(* CODESYS project PCL_CoralP

Project tree, tasks and I/O mapping:
  Device : CODESYS Control for Linux SL, CODESYS, order no. 2302000005, version 4.11.0.0
    Ethernet : Ethernet, CODESYS, version 4.2.0.0
        settings: IPAddress = [172,16,0,11]; SubnetMask = [205,255,255,0]; GatewayAddress = [0,0,0,0]; MACAddress = [16#00,16#E0,16#4F,16#68,16#EC,16#4A]; NetworkInterfaceName = 'eno1'; NetworkInterfaceName = "eno1"; SaveCommunicationSettings = FALSE; IPAddress = [192,168,0,2]; SubnetMask = [255,255,255,0]; GatewayAddress = [0,0,0,0]
      Modbus_TCP_Master : Modbus TCP Master, 3S - Smart Software Solutions GmbH, version 4.3.0.0 (disabled)
          settings: AutoReconnect = TRUE
        Modbus_TCP_Slave_AC1 : Modbus TCP Slave, 3S - Smart Software Solutions GmbH, version 4.1.0.0
            settings: Unit-ID = 255; IPAddress = [192, 168, 0, 51]; Channel 0.Function Code = 3; Channel 0.Read Offset = 16#0000; Channel 0.Read Length = 124; Channel 0.Write Offset = 0; Channel 0.Write Length = 0; Channel 0.Cycle Time = 100; Channel 1.Function Code = 3; Channel 1.Read Offset = 16#007C; Channel 1.Read Length = 124; Channel 1.Write Offset = 0; Channel 1.Write Length = 0; Channel 1.Cycle Time = 100; Channel 2.Function Code = 3; Channel 2.Read Offset = 16#00F8; Channel 2.Read Length = 124; Channel 2.Write Offset = 0; Channel 2.Write Length = 0; Channel 2.Cycle Time = 100; Channel 3.Function Code = 16; Channel 3.Read Offset = 0; Channel 3.Read Length = 0; Channel 3.Write Offset = 16#0114; Channel 3.Write Length = 4; Channel 3.Cycle Time = 100
            output Application.Chiller_1.modbus_var_1002[276] : WORD  // Channel 3.Channel 3
            output Application.Chiller_1.modbus_var_1002[277] : WORD  // Channel 3.Channel 3
            output Application.Chiller_1.modbus_var_1002[278] : WORD  // Channel 3.Channel 3
            output Application.Chiller_1.modbus_var_1002[279] : WORD  // Channel 3.Channel 3
            unmapped channels: Channel 0, Channel 1, Channel 2, Channel 3
  Modbus_Master_COM_Port_1 : Modbus Master, COM Port, 3S - Smart Software Solutions GmbH, version 4.3.0.0
      settings: Auto-restart communication = TRUE
    Modbus_Server_COM_Port_AC1 : Modbus Server, COM Port, CODESYS, version 4.4.0.0
        settings: SlaveAddress = 18; ResponseTimeout = 1000; UseExtendedFunctionCodes = TRUE; Channel 0.Function Code = 3; Channel 0.Read Offset = 16#0000; Channel 0.Read Length = 91; Channel 0.Write Offset = 0; Channel 0.Write Length = 0; Channel 0.Cycle Time = 100
        input  Application.Chiller_1.modbus_var_1000 : ARRAY[0..90] OF WORD  // Channel 0
    Modbus_Server_COM_Port_AC2 : Modbus Server, COM Port, CODESYS, version 4.4.0.0
        settings: SlaveAddress = 18; ResponseTimeout = 1000; UseExtendedFunctionCodes = TRUE; Channel 0.Function Code = 3; Channel 0.Read Offset = 16#0000; Channel 0.Read Length = 91; Channel 0.Write Offset = 0; Channel 0.Write Length = 0; Channel 0.Cycle Time = 100
        input  Application.Chiller_2.modbus_var_1000 : ARRAY[0..90] OF WORD  // Channel 0
    Modbus_Slave_COM_Port_AC1 : Modbus Slave, COM Port, 3S - Smart Software Solutions GmbH, version 4.1.0.0
        settings: SlaveAddress = 18; ResponseTimeout = 1000; UseExtendedFunctionCodes = TRUE; Channel 0.Function Code = 3; Channel 0.Read Offset = 16#0000; Channel 0.Read Length = 100; Channel 0.Write Offset = 0; Channel 0.Write Length = 0; Channel 0.Cycle Time = 100
        input  Application.Chiller_1.modbus_var_1000 : ARRAY[0..99] OF WORD  // Channel 0
    Modbus_Slave_COM_Port_AC2 : Modbus Slave, COM Port, 3S - Smart Software Solutions GmbH, version 4.1.0.0
        settings: SlaveAddress = 18; ResponseTimeout = 1000; UseExtendedFunctionCodes = TRUE; Channel 0.Function Code = 3; Channel 0.Read Offset = 16#0200; Channel 0.Read Length = 91; Channel 0.Write Offset = 0; Channel 0.Write Length = 0; Channel 0.Cycle Time = 100
        input  Application.Chiller_2.modbus_var_1000 : ARRAY[0..90] OF WORD  // Channel 0
    Modbus_Slave_COM_Port_AC3 : Modbus Slave, COM Port, 3S - Smart Software Solutions GmbH, version 4.1.0.0
        settings: SlaveAddress = 18; ResponseTimeout = 1000; UseExtendedFunctionCodes = TRUE; Channel 0.Function Code = 3; Channel 0.Read Offset = 16#0400; Channel 0.Read Length = 91; Channel 0.Write Offset = 0; Channel 0.Write Length = 0; Channel 0.Cycle Time = 100
        input  Application.Chiller_3.modbus_var_1000 : ARRAY[0..90] OF WORD  // Channel 0
    Modbus_Slave_COM_Port_AC4 : Modbus Slave, COM Port, 3S - Smart Software Solutions GmbH, version 4.1.0.0
        settings: SlaveAddress = 18; ResponseTimeout = 1000; UseExtendedFunctionCodes = TRUE; Channel 0.Function Code = 3; Channel 0.Read Offset = 16#0600; Channel 0.Read Length = 91; Channel 0.Write Offset = 0; Channel 0.Write Length = 0; Channel 0.Cycle Time = 100
        input  Application.Chiller_4.modbus_var_1000 : ARRAY[0..90] OF WORD  // Channel 0
    Modbus_Slave_COM_Seq : Modbus Slave, COM Port, 3S - Smart Software Solutions GmbH, version 4.1.0.0
        settings: SlaveAddress = 18; ResponseTimeout = 1000; UseExtendedFunctionCodes = TRUE; Channel 0.Function Code = 3; Channel 0.Read Offset = 16#0A00; Channel 0.Read Length = 125; Channel 0.Write Offset = 0; Channel 0.Write Length = 0; Channel 0.Cycle Time = 100; Channel 1.Function Code = 3; Channel 1.Read Offset = 16#0A7D; Channel 1.Read Length = 34; Channel 1.Write Offset = 0; Channel 1.Write Length = 0; Channel 1.Cycle Time = 100; Channel 2.Function Code = 16; Channel 2.Read Offset = 0; Channel 2.Read Length = 0; Channel 2.Write Offset = 16#0A8B; Channel 2.Write Length = 4; Channel 2.Cycle Time = 100; Channel 3.Function Code = 16; Channel 3.Read Offset = 0; Channel 3.Read Length = 0; Channel 3.Write Offset = 16#0A95; Channel 3.Write Length = 4; Channel 3.Cycle Time = 100
        input  Application.Sequence.modbus_var_1000 : ARRAY[0..124] OF WORD  // Channel 0
        input  Application.Sequence.modbus_var_1001 : ARRAY[0..33] OF WORD  // Channel 1
        output Application.Sequence.modbus_var_PI : ARRAY[0..3] OF WORD  // Channel 2
        output Application.Sequence.modbus_var_wasted : ARRAY[0..3] OF WORD  // Channel 3
  libraries: CmpBitmapPool, 3.5.17.0 (System); AC_DataLog, 3.5.16.0 (3S - Smart Software Solutions GmbH)
  5ce3da45-db07-42e7-a21c-a00fff4ed8f6|C:\Users\Codesys\Desktop\Images\Div bilder\Arrow gray left.png
  5ce3da45-db07-42e7-a21c-a00fff4ed8f6|C:\Users\Codesys\Desktop\Images\Div bilder\Arrow green down.png
  5ce3da45-db07-42e7-a21c-a00fff4ed8f6|C:\Users\Codesys\Desktop\Images\Div bilder\Arrow green up.png
  5ce3da45-db07-42e7-a21c-a00fff4ed8f6|C:\Users\Codesys\Desktop\Images\Div bilder\Arrow lightblue left.png
  5ce3da45-db07-42e7-a21c-a00fff4ed8f6|C:\Users\Codesys\Desktop\Images\Div bilder\Arrow red down.png
  5ce3da45-db07-42e7-a21c-a00fff4ed8f6|C:\Users\Codesys\Desktop\Images\Div bilder\Arrow red left.png
  5ce3da45-db07-42e7-a21c-a00fff4ed8f6|C:\Users\Codesys\Desktop\Images\Invisible.png
  5ce3da45-db07-42e7-a21c-a00fff4ed8f6|C:\Users\Codesys\Desktop\Images\LEDS\ALARM.png
  5ce3da45-db07-42e7-a21c-a00fff4ed8f6|C:\Users\Codesys\Desktop\Images\LEDS\Led_SQ_Green1_On_Medium.png
  5ce3da45-db07-42e7-a21c-a00fff4ed8f6|C:\Users\Codesys\Desktop\Images\LEDS\Led_SQ_Grey_Off_Medium.png
  5ce3da45-db07-42e7-a21c-a00fff4ed8f6|C:\Users\Codesys\Desktop\Images\LEDS\TRIP.png
  5ce3da45-db07-42e7-a21c-a00fff4ed8f6|C:\Users\Codesys\Desktop\Images\Logo-Aida.png
  5ce3da45-db07-42e7-a21c-a00fff4ed8f6|C:\Users\Codesys\Desktop\Images\Logo-Costa.png
  5ce3da45-db07-42e7-a21c-a00fff4ed8f6|C:\Users\Codesys\Desktop\Images\Logo-HAL.png
  5ce3da45-db07-42e7-a21c-a00fff4ed8f6|C:\Users\Codesys\Desktop\Images\Logo-ncl.png
  5ce3da45-db07-42e7-a21c-a00fff4ed8f6|C:\Users\Codesys\Desktop\Images\Logo-Princess.png
  5ce3da45-db07-42e7-a21c-a00fff4ed8f6|C:\Users\Codesys\Desktop\Images\Logo-TUI.png
  5ce3da45-db07-42e7-a21c-a00fff4ed8f6|C:\Users\Codesys\Desktop\Images\Menu\AlarmMenu.png
  5ce3da45-db07-42e7-a21c-a00fff4ed8f6|C:\Users\Codesys\Desktop\Images\Pipes\PipeGreen_1_Horizontal.png
  5ce3da45-db07-42e7-a21c-a00fff4ed8f6|C:\Users\Codesys\Desktop\Images\Pipes\PipeGreen_1_LD.png
  5ce3da45-db07-42e7-a21c-a00fff4ed8f6|C:\Users\Codesys\Desktop\Images\Pipes\PipeGreen_2_LU.png
  5ce3da45-db07-42e7-a21c-a00fff4ed8f6|C:\Users\Codesys\Desktop\Images\Pipes\PipeGreen_3way_2.png
  5ce3da45-db07-42e7-a21c-a00fff4ed8f6|C:\Users\Codesys\Desktop\Images\Pipes\PipeGreen_3way.png
  5ce3da45-db07-42e7-a21c-a00fff4ed8f6|C:\Users\Codesys\Desktop\Images\Pipes\PipeGrey_1S_Horizontal.png
  5ce3da45-db07-42e7-a21c-a00fff4ed8f6|C:\Users\Codesys\Desktop\Images\Pipes\PipeGrey_2_LD.png
  5ce3da45-db07-42e7-a21c-a00fff4ed8f6|C:\Users\Codesys\Desktop\Images\Pipes\PipeGrey_3_LU.png
  5ce3da45-db07-42e7-a21c-a00fff4ed8f6|C:\Users\Codesys\Desktop\Images\Pipes\PipeLightBlue_1_Horizontal.png
  5ce3da45-db07-42e7-a21c-a00fff4ed8f6|C:\Users\Codesys\Desktop\Images\Pipes\PipeLightBlue_1_LD.png
  5ce3da45-db07-42e7-a21c-a00fff4ed8f6|C:\Users\Codesys\Desktop\Images\Pipes\PipeLightBlue_1_Vertical.png
  5ce3da45-db07-42e7-a21c-a00fff4ed8f6|C:\Users\Codesys\Desktop\Images\Pipes\PipeLightBlue_2_LU.png
  5ce3da45-db07-42e7-a21c-a00fff4ed8f6|C:\Users\Codesys\Desktop\Images\Pipes\PipeLightBlue_3_RD.png
  5ce3da45-db07-42e7-a21c-a00fff4ed8f6|C:\Users\Codesys\Desktop\Images\Pipes\PipeLightBlue_3_RU.png
  5ce3da45-db07-42e7-a21c-a00fff4ed8f6|C:\Users\Codesys\Desktop\Images\Pipes\PipeRed_1_LD.png
  5ce3da45-db07-42e7-a21c-a00fff4ed8f6|C:\Users\Codesys\Desktop\Images\Pipes\PipeRed_1_RD.png
  5ce3da45-db07-42e7-a21c-a00fff4ed8f6|C:\Users\Codesys\Desktop\Images\Pipes\PipeRed_2_Horizontal.png
  5ce3da45-db07-42e7-a21c-a00fff4ed8f6|C:\Users\Codesys\Desktop\Images\Pipes\PipeRed_2_LU.png
  5ce3da45-db07-42e7-a21c-a00fff4ed8f6|C:\Users\Codesys\Desktop\Images\Pipes\PipeRed_2_RU.png
  5ce3da45-db07-42e7-a21c-a00fff4ed8f6|C:\Users\Codesys\Desktop\Images\Pumps\Pump_Large_3.png
  5ce3da45-db07-42e7-a21c-a00fff4ed8f6|C:\Users\Codesys\Desktop\Images\Scales\BarScale3.png
  5ce3da45-db07-42e7-a21c-a00fff4ed8f6|C:\Users\Codesys\Desktop\Images\Scales\BarScale4.png
  5ce3da45-db07-42e7-a21c-a00fff4ed8f6|C:\Users\Codesys\Desktop\Images\Transparants\CapBarTranparant.png
  5ce3da45-db07-42e7-a21c-a00fff4ed8f6|C:\Users\Codesys\Desktop\Images\Valves\Valve_2.png
  5ce3da45-db07-42e7-a21c-a00fff4ed8f6|C:\Users\Codesys\Desktop\Images\Valves\Valve_3.png
  5ce3da45-db07-42e7-a21c-a00fff4ed8f6|C:\Users\Codesys\Desktop\Images\Valves\Valve_4.png
  5ce3da45-db07-42e7-a21c-a00fff4ed8f6|C:\Users\Codesys\Desktop\MenuAlarm.png
  5ce3da45-db07-42e7-a21c-a00fff4ed8f6|C:\Users\Codesys\Desktop\MenuEvents.png
  5ce3da45-db07-42e7-a21c-a00fff4ed8f6|C:\Users\Codesys\Desktop\MenuHome.png
  5ce3da45-db07-42e7-a21c-a00fff4ed8f6|C:\Users\Codesys\Desktop\MenuLogout.png
  5ce3da45-db07-42e7-a21c-a00fff4ed8f6|C:\Users\Codesys\Desktop\MenuSchematics.png
  5ce3da45-db07-42e7-a21c-a00fff4ed8f6|C:\Users\Codesys\Desktop\MenuSettings.png
  5ce3da45-db07-42e7-a21c-a00fff4ed8f6|C:\Users\Codesys\Desktop\white.PNG
  5ce3da45-db07-42e7-a21c-a00fff4ed8f6|C:\Users\Codesys\Documents\logo\1200px-Johnson_Controls.svg.png
  5ce3da45-db07-42e7-a21c-a00fff4ed8f6|C:\Users\Codesys\Documents\logo\JCI_Full Color_Transparent Background.png
  5ce3da45-db07-42e7-a21c-a00fff4ed8f6|C:\Users\Codesys\Pictures\ConquestVSChiller1.jpg
  5ce3da45-db07-42e7-a21c-a00fff4ed8f6|C:\Users\Codesys\Pictures\Grafic_oldradar\2016_update\Images\Chiller\Compressor.png
  5ce3da45-db07-42e7-a21c-a00fff4ed8f6|C:\Users\Codesys\Pictures\Grafic_oldradar\2016_update\Images\Chiller\Condenser.png
  5ce3da45-db07-42e7-a21c-a00fff4ed8f6|C:\Users\Codesys\Pictures\Grafic_oldradar\2016_update\Images\Chiller\Evaporator.png
  5ce3da45-db07-42e7-a21c-a00fff4ed8f6|C:\Users\Technician\Desktop\Images\Pipes\PipeBlack_1_Vertical.png
  5ce3da45-db07-42e7-a21c-a00fff4ed8f6|C:\Users\Technician\Desktop\Images\Ships\CoralP.jpg
  5ce3da45-db07-42e7-a21c-a00fff4ed8f6|C:\Users\Technician\Desktop\Images\Ships\Diamond.png
  5ce3da45-db07-42e7-a21c-a00fff4ed8f6|C:\Users\Technician\Pictures\C_Sunrise.jpg
  5ce3da45-db07-42e7-a21c-a00fff4ed8f6|C:\Users\Technician\Pictures\Sapphire-princess.jpg
  5ce3da45-db07-42e7-a21c-a00fff4ed8f6|E:\Images\Images\Chiller\ACChiller3D.png
  text list GlobalTextList
  visualisation AC_Plant_Overview
  Alarm Configuration
  visualisation Alarm_list
  program BlinkingAlarm [CFC]
  program Calculus [ST]
  visualisation Chiller1Menu
  visualisation Chiller2Menu
  visualisation Chiller3Menu
  visualisation Chiller4Menu
  program Chiller_1 [ST]
  visualisation Chiller_1_Alarm
  visualisation Chiller_1_Alarm
  visualisation Chiller_1_Flow_Diagram
  visualisation Chiller_1_Oil
  text list Chiller_1_trendvalues
  visualisation Chiller_1_Trip
  visualisation Chiller_1_Trip
  visualisation Chiller_1_Values
  visualisation Chiller_1_Values
  visualisation Chiller_1_VFD
  program Chiller_2 [ST]
  text list Chiller_2_4_trendvalues
  visualisation Chiller_2_Alarm
  visualisation Chiller_2_Alarm
  visualisation Chiller_2_Flow_Diagram
  visualisation Chiller_2_Flow_Diagram
  visualisation Chiller_2_Oil
  visualisation Chiller_2_Trip
  visualisation Chiller_2_Trip
  visualisation Chiller_2_Values
  visualisation Chiller_2_Values
  visualisation Chiller_3_Alarm
  program Chiller_3 [ST]
  visualisation Chiller_3_Flow_Diagram
  visualisation Chiller_3_Flow_Diagram
  visualisation Chiller_3_Oil
  text list Chiller_3_trendvalues
  visualisation Chiller_3_Trip
  program Chiller_4 [ST]
  visualisation Chiller_4_Alarm
  visualisation Chiller_4_Alarm
  visualisation Chiller_4_Oil
  text list Chiller_4_trendvalues
  global variables GVL
  text PersistenceConfig
  text list Sequence_trendvalues
  function block AC_DataLogManager [ST]
*)

// GVL
{attribute 'qualified_only'}
VAR_GLOBAL
	COPcalc_data	: ARRAY[0..2, 0..320] OF STRING(100);
	calc_data		: ARRAY[0..8, 0..80] OF STRING(100) ;
	{attribute 'ac_persist' := 'PersistenceChannel'}
	saCOPDataArray			: ARRAY[0..2, 0..320] OF STRING(100);
	{attribute 'ac_persist' := 'PersistenceChannel'}
	saDataArray			: ARRAY[0..8, 0..80] OF STRING(100);
		{attribute 'ac_persist' := 'PersistenceChannel'}
	saDataArray1			: ARRAY[0..8, 0..80] OF STRING(100);
		{attribute 'ac_persist' := 'PersistenceChannel'}
	saDataArray2		: ARRAY[0..8, 0..80] OF STRING(100);
	initRead : BOOL;
	xRead : BOOL;
	xRead1 : BOOL;
	xRead2 : BOOL;
	xReadCOP : BOOL := FALSE;
	startUp : BOOL;
	presstimer  : TON;
	presstimer2 : TON;
	presstimer3 : TON;
	presstimer4 : TON;
	delaytimer  : TON;
	starttimer1 : BOOL := FALSE  ;
	starttimer2 : BOOL := FALSE  ;
	starttimer3 : BOOL := FALSE  ;
	starttimer4 : BOOL := FALSE  ;
	startdelaytimer : BOOL := FALSE ;
	Startonce : BOOL := FALSE ;
	Startsecond : BOOL := FALSE ;
	{attribute 'ac_persist' := 'PersistenceChannel'}
	PIexpireDate : DATE_AND_TIME := DT#2025-12-30-00:00:00;
	CurrentDate : DATE_AND_TIME ;
	
	
END_VAR

// BlinkingAlarm
PROGRAM BlinkingAlarm
VAR
	TimeOn: TIME:= T#1S;
	TimeOff: TIME:= T#1S;
	Alarm: BOOL;
	TurnOn: BOOL;
		
	Blink_0: BLINK;
	
END_VAR
VAR // added by the converter: edge detectors and wires of the graphical bodies
    _w1, _w2 : BOOL;
END_VAR

TurnOn := _w1;
_w1 := not.Sequence.Alarm_sequence OR not.Chiller_1.Unit_alarm OR not.Chiller_1.Unit_trip OR not.Chiller_2.Unit_alarm OR not.Chiller_2.Unit_trip OR not.Chiller_3.Unit_alarm OR not.Chiller_3.Unit_trip OR not.Chiller_4.Unit_alarm OR not.Chiller_4.Unit_trip;
_w2 := TurnOn AND Blink_0.OUT;
Blink_0(ENABLE := TurnOn, TIMELOW := TimeOff, TIMEHIGH := TimeOn); // BLINK
Alarm := _w2;

END_PROGRAM

// Chiller_2
PROGRAM Chiller_2
VAR

timer2 : standard.ton ;
{attribute 'ac_datalog_set_default_group' := 'DatalogChannel_2'}
instStruct : LogStruct;

modbus_var : ARRAY[0..100] OF INT;
modbus_var_1000 : ARRAY[0..123] OF WORD;
modbus_var_1001 : ARRAY[124..247] OF WORD;
modbus_var_1002 : ARRAY[248..371] OF WORD;
{attribute 'ac_datalog_hysteresis' := '0.2'}
{attribute 'ac_datalog' := 'DatalogChannel_2'}
Temp_chilled_medium_out : REAL;
{attribute 'ac_datalog_hysteresis' := '0.2'}
{attribute 'ac_datalog' := 'DatalogChannel_2'}
Temp_chilled_medium_in : REAL;
{attribute 'ac_datalog_hysteresis' := '0.2'}
{attribute 'ac_datalog' := 'DatalogChannel_2'}
Temp_water_inlet_cond : REAL;
{attribute 'ac_datalog_hysteresis' := '0.2'}
{attribute 'ac_datalog' := 'DatalogChannel_2'}
Press_suction_compr : REAL;
{attribute 'ac_datalog_hysteresis' := '0.5'}
{attribute 'ac_datalog' := 'DatalogChannel_2'}
Press_discharge_compr : REAL;
{attribute 'ac_datalog_hysteresis' := '0.5'}
{attribute 'ac_datalog' := 'DatalogChannel_2'}
Press_oil_receiver : REAL;
{attribute 'ac_datalog_hysteresis' := '0.5'}
{attribute 'ac_datalog' := 'DatalogChannel_2'}
Press_oil_compr : REAL;
{attribute 'ac_datalog_hysteresis' := '0.4'}
{attribute 'ac_datalog' := 'DatalogChannel_2'}
Temp_discharge : REAL;
{attribute 'ac_datalog_hysteresis' := '0.5'}
{attribute 'ac_datalog' := 'DatalogChannel_2'}
Oil_temp_receiver : REAL;
{attribute 'ac_datalog_hysteresis' := '0.5'}
{attribute 'ac_datalog' := 'DatalogChannel_2'}
Max_motor_temp : REAL;
{attribute 'ac_datalog_hysteresis' := '0.2'}
{attribute 'ac_datalog' := 'DatalogChannel_2'}
Temp_motor_bearing_DE : REAL;
{attribute 'ac_datalog_hysteresis' := '0.2'}
{attribute 'ac_datalog' := 'DatalogChannel_2'}
Temp_motor_bearing_NDE : REAL;
{attribute 'ac_datalog_hysteresis' := '4'}
{attribute 'ac_datalog' := 'DatalogChannel_2'}
Motor_current : REAL;
{attribute 'ac_datalog_hysteresis' := '50'}
{attribute 'ac_datalog' := 'DatalogChannel_2'}
Running_hours_comp_unscaled : WORD;
{attribute 'ac_datalog_hysteresis' := '50'}
{attribute 'ac_datalog' := 'DatalogChannel_2'}
Running_hours_oil_pump_unscaled : WORD;
{attribute 'ac_datalog' := 'DatalogChannel_2'}
Anti_recycle_time : REAL;
{attribute 'ac_datalog_hysteresis' := '2'}
{attribute 'ac_datalog' := 'DatalogChannel_2'}
Feedback_compressor : REAL;
{attribute 'ac_datalog_hysteresis' := '0.2'}
{attribute 'ac_datalog' := 'DatalogChannel_2'}
Oil_diff_pressure : REAL;
{attribute 'ac_datalog_hysteresis' := '0.3'}
{attribute 'ac_datalog' := 'DatalogChannel_2'}
Suction_saturated_temp : REAL;
{attribute 'ac_datalog_hysteresis' := '0.2'}
{attribute 'ac_datalog' := 'DatalogChannel_2'}
Discharge_saturated_temp : REAL;
{attribute 'ac_datalog_hysteresis' := '0.2'}
{attribute 'ac_datalog' := 'DatalogChannel_2'}
Temp_water_outlet_cond : REAL;
{attribute 'ac_datalog_hysteresis' := '0.2'}
{attribute 'ac_datalog' := 'DatalogChannel_2'}
Temp_motor_wind_R : REAL;
{attribute 'ac_datalog_hysteresis' := '0.2'}
{attribute 'ac_datalog' := 'DatalogChannel_2'}
Temp_motor_wind_S : REAL;
{attribute 'ac_datalog_hysteresis' := '0.2'}
{attribute 'ac_datalog' := 'DatalogChannel_2'}
Temp_motor_wind_T : REAL;
{attribute 'ac_datalog_hysteresis' := '0.2'}
{attribute 'ac_datalog' := 'DatalogChannel_2'}
Temp_motor_air : REAL;
{attribute 'ac_datalog_hysteresis' := '0.04'}
{attribute 'ac_datalog' := 'DatalogChannel_2'}
dP_CW : REAL;
{attribute 'ac_datalog_hysteresis' := '0.04'}
{attribute 'ac_datalog' := 'DatalogChannel_2'}
dP_SW : REAL;
{attribute 'ac_datalog_hysteresis' := '4'}
{attribute 'ac_datalog' := 'DatalogChannel_2'}
Chiller_capacity : REAL;
{attribute 'ac_datalog_hysteresis' := '2'}
{attribute 'ac_datalog' := 'DatalogChannel_2'}
Temp_oil_inlet_compr : REAL;
Spare : REAL;
{attribute 'ac_datalog_hysteresis' := '2'}
{attribute 'ac_datalog' := 'DatalogChannel_2'}
SP_CW_controller : REAL;
{attribute 'ac_datalog_hysteresis' := '2'}
{attribute 'ac_datalog' := 'DatalogChannel_2'}
Setpoint_oil_pump : REAL;
{attribute 'ac_datalog_hysteresis' := '0.02'}
{attribute 'ac_datalog' := 'DatalogChannel_2'}
Thrust_bearing_position : REAL;
{attribute 'ac_datalog_hysteresis' := '50'}
{attribute 'ac_datalog' := 'DatalogChannel_2'}
Oil_pump_running_hours : REAL;
{attribute 'ac_datalog_hysteresis' := '5'}
{attribute 'ac_datalog' := 'DatalogChannel_2'}
Liquid_level_condenser : REAL;
{attribute 'ac_datalog_hysteresis' := '0.05'}
{attribute 'ac_datalog' := 'DatalogChannel_2'}
Oil_Filter_Drop : REAL; 
{attribute 'ac_datalog_hysteresis' := '2'}
{attribute 'ac_datalog' := 'DatalogChannel_2'}
Proximitor_thrust_pos : REAL;
{attribute 'ac_datalog_hysteresis' := '0.4'}
{attribute 'ac_datalog' := 'DatalogChannel_2'}
Press_chilled_medium_in : REAL;
{attribute 'ac_datalog_hysteresis' := '0.2'}
{attribute 'ac_datalog' := 'DatalogChannel_2'}
Press_water_cond_out : REAL;
{attribute 'ac_datalog_hysteresis' := '0.02'}
{attribute 'ac_datalog' := 'DatalogChannel_2'}
Feedback_sea_water_valve : REAL;
{attribute 'ac_datalog_hysteresis' := '1'}
{attribute 'ac_datalog' := 'DatalogChannel_2'}
Oil_pressure_before_filter : REAL;
{attribute 'ac_datalog_hysteresis' := '0.2'}
{attribute 'ac_datalog' := 'DatalogChannel_2'}
Trafo_winding_temp : REAL;
{attribute 'ac_datalog_hysteresis' := '1'}
{attribute 'ac_datalog' := 'DatalogChannel_2'}
Feedback_VGD : REAL;
{attribute 'ac_datalog_hysteresis' := '4'}
{attribute 'ac_datalog' := 'DatalogChannel_2'}
Feedback_liquid_valve : REAL;
{attribute 'ac_datalog_hysteresis' := '3'}
{attribute 'ac_datalog' := 'DatalogChannel_2'}
Feedback_HGV : REAL;
{attribute 'ac_datalog_hysteresis' := '2'}
{attribute 'ac_datalog' := 'DatalogChannel_2'}
Discharge_superheat : REAL;
{attribute 'ac_datalog_hysteresis' := '0.6'}
{attribute 'ac_datalog' := 'DatalogChannel_2'}
Frequency_oil_pump : REAL;
{attribute 'ac_datalog_hysteresis' := '3'}
{attribute 'ac_datalog' := 'DatalogChannel_2'}
Hot_gas_valve_output : REAL;
{attribute 'ac_datalog_hysteresis' := '2'}
{attribute 'ac_datalog' := 'DatalogChannel_2'}
Control_signal_unit_d : REAL;
{attribute 'ac_datalog_hysteresis' := '2'}
{attribute 'ac_datalog' := 'DatalogChannel_2'}
Stall_detector : REAL;
{attribute 'ac_datalog_hysteresis' := '0.2'}
{attribute 'ac_datalog' := 'DatalogChannel_2'}
SP_MC_controller : REAL;
{attribute 'ac_datalog_hysteresis' := '2'}
{attribute 'ac_datalog' := 'DatalogChannel_2'}
Prerotary_output : REAL;
{attribute 'ac_datalog_hysteresis' := '2'}
{attribute 'ac_datalog' := 'DatalogChannel_2'}
VGD_output : REAL;
{attribute 'ac_datalog_hysteresis' := '2'}
{attribute 'ac_datalog' := 'DatalogChannel_2'}
SP_PID_compressor : REAL;
{attribute 'ac_datalog_hysteresis' := '2'}
{attribute 'ac_datalog' := 'DatalogChannel_2'}
Output_PID_suction : REAL;
{attribute 'ac_datalog_hysteresis' := '2'}
{attribute 'ac_datalog' := 'DatalogChannel_2'}
Output_PID_discharge : REAL;
{attribute 'ac_datalog_hysteresis' := '2'}
{attribute 'ac_datalog' := 'DatalogChannel_2'}
Output_PID_motor : REAL;
{attribute 'ac_datalog_hysteresis' := '2'}
{attribute 'ac_datalog' := 'DatalogChannel_2'}
Output_PID_superheat : REAL;
{attribute 'ac_datalog_hysteresis' := '2'}
{attribute 'ac_datalog' := 'DatalogChannel_2'}
SP_control : REAL;
{attribute 'ac_datalog_hysteresis' := '2'}
{attribute 'ac_datalog' := 'DatalogChannel_2'}
Unit_control_signal : REAL;
{attribute 'ac_datalog_hysteresis' := '2'}
{attribute 'ac_datalog' := 'DatalogChannel_2'}
Feedback_PRV : REAL;
{attribute 'ac_datalog_hysteresis' := '0.3'}
{attribute 'ac_datalog' := 'DatalogChannel_2'}
Theta_out : REAL;
{attribute 'ac_datalog_hysteresis' := '50'}
{attribute 'ac_datalog' := 'DatalogChannel_2'}
Alarm_limit_stall_count_unscaled : WORD;
{attribute 'ac_datalog_hysteresis' := '50'}
{attribute 'ac_datalog' := 'DatalogChannel_2'}
Alarm_limit_stall_count : REAL;
{attribute 'ac_datalog_hysteresis' := '2'}
{attribute 'ac_datalog' := 'DatalogChannel_2'}
Stall_ramp : REAL;
Min_allowed_PRVposition : REAL;
Number_of_starts : REAL;
SP_freq_oil_pump_VFD : REAL;
SP_oil_pressure_diff : REAL;
SP_oil_pressure : REAL;
{attribute 'ac_datalog_hysteresis' := '2'}
{attribute 'ac_datalog' := 'DatalogChannel_2'}
Setpoint_conv_oil_pump : REAL;
Days_above_stall_limit : REAL;
Hrs_above_stall_limit : REAL;
Min_above_stall_limit : REAL;
Sec_above_stall_limit : REAL;
{attribute 'ac_datalog_hysteresis' := '2'}
{attribute 'ac_datalog' := 'DatalogChannel_2'}
SP_cond_press : REAL;
{attribute 'ac_datalog_hysteresis' := '2'}
{attribute 'ac_datalog' := 'DatalogChannel_2'}
SP_PID_Level : REAL;
{attribute 'ac_datalog_hysteresis' := '2'}
{attribute 'ac_datalog' := 'DatalogChannel_2'}
Control_signal_SW_valve : REAL;
{attribute 'ac_datalog_hysteresis' := '4'}
{attribute 'ac_datalog' := 'DatalogChannel_2'}
Liquid_valve_output : REAL;
{attribute 'ac_datalog_hysteresis' := '0.2'}
{attribute 'ac_datalog' := 'DatalogChannel_2'}
SP_PID_seawater : REAL;
{attribute 'ac_datalog_hysteresis' := '4'}
{attribute 'ac_datalog' := 'DatalogChannel_2'}
Chiller_capacity_t1 : REAL;
{attribute 'ac_datalog_hysteresis' := '2'}
{attribute 'ac_datalog' := 'DatalogChannel_2'}
SW_pump_speed_order : REAL;
{attribute 'ac_datalog_hysteresis' := '0.4'}
{attribute 'ac_datalog' := 'DatalogChannel_2'}
Press_chilled_medium_out : REAL;
{attribute 'ac_datalog_hysteresis' := '50'}
{attribute 'ac_datalog' := 'DatalogChannel_2'}
Running_hours_compressormotor : REAL;
{attribute 'ac_datalog_hysteresis' := '0.2'}
{attribute 'ac_datalog' := 'DatalogChannel_2'}
Press_water_cond_inlet : REAL;
{attribute 'ac_datalog_hysteresis' := '2'}
{attribute 'ac_datalog' := 'DatalogChannel_2'}
Speed_feedback_VFD : REAL;
{attribute 'ac_datalog_hysteresis' := '2'}
{attribute 'ac_datalog' := 'DatalogChannel_2'}
Order_VFD_perc : REAL;
{attribute 'ac_datalog_hysteresis' := '2'}
{attribute 'ac_datalog' := 'DatalogChannel_2'}
Order_VFD_Hz : REAL;
{attribute 'ac_datalog_hysteresis' := '2'}
{attribute 'ac_datalog' := 'DatalogChannel_2'}
Temp_trafo_wind_U : REAL;
{attribute 'ac_datalog_hysteresis' := '0.2'}
{attribute 'ac_datalog' := 'DatalogChannel_2'}
Temp_trafo_wind_V : REAL;
{attribute 'ac_datalog_hysteresis' := '0.2'}
{attribute 'ac_datalog' := 'DatalogChannel_2'}
Temp_trafo_wind_W : REAL;
{attribute 'ac_datalog_hysteresis' := '2'}
{attribute 'ac_datalog' := 'DatalogChannel_2'}
Opt_speed_VFD_perc : REAL;
{attribute 'ac_datalog_hysteresis' := '2'}
{attribute 'ac_datalog' := 'DatalogChannel_2'}
Opt_speed_VFD_Hz : REAL;
Surge_counter_VFD : REAL;
Spare_4 : REAL;
Spare_3 : REAL;
Spare_2 : REAL;
Spare_0 : REAL;
Vibration_compressor_DE: REAL;
Vibration_compressor_NDE: REAL;
Feedback_seawater_valve_overboard : REAL;
Feedback_seawater_valve_bypass : REAL;
CW_flow_m3: REAL;
SW_flow_m3: REAL;
Max_motor_wind_temp: REAL;
Order_SWW_overboard: REAL;
Order_SWW_bypass: REAL;
{attribute 'ac_datalog_hysteresis' := '0.4'}
{attribute 'ac_datalog' := 'DatalogChannel'}
COP_chiller_mech : REAL ;
{attribute 'ac_datalog_hysteresis' := '50'}
{attribute 'ac_datalog' := 'DatalogChannel'}
P2_mot_1_kW : REAL ;
{attribute 'ac_datalog_hysteresis' := '50'}
{attribute 'ac_datalog' := 'DatalogChannel'}
P1_motor_kW : REAL ;
{attribute 'ac_datalog_hysteresis' := '0.4'}
{attribute 'ac_datalog' := 'DatalogChannel'}
COP_chiller_ele : REAL ;
{attribute 'ac_datalog_hysteresis' := '0.2'}
{attribute 'ac_datalog' := 'DatalogChannel'}
PI_chiller : REAL ;
;{attribute 'ac_datalog_hysteresis' := '40'}
{attribute 'ac_datalog' := 'DatalogChannel'}
Wasted_energy_kW : REAL ;
{attribute 'ac_datalog_hysteresis' := '200'}
{attribute 'ac_datalog' := 'DatalogChannel'}
Chiller_capacity_kW : REAL;
Thrust_bearing_ref_min : REAL ;
Thrust_bearing_ref_max : REAL ;
Thrust_bearing_ref : REAL ;
Q2_chillerMWh : REAL ;
Chiller_P1_MWh : REAL ;
Cal_date_MMYY : REAL ;
Chiller_P2_MWh : REAL ;
Liquid_line_temp : REAL ;
VFD_motor_current : REAL ;
Feedback_liquid_valve_raw : REAL ;
Feedback_VGD_raw : REAL ;
Feedback_PRV_raw : REAL ;
Feedback_HGV_raw : REAL ;
Feedback_seawater_valve_overboard_raw : REAL ;
Feedback_seawater_valve_bypass_raw : REAL ;
SP_cond_press_limit : REAL ;
SP_evap_press_limit : REAL ;
SP_discharge_superheat_limit : REAL ;
SP_t1 : REAL ;
VFD_min_allowed_frequence : REAL ;
VFD_min_allowed_speed : REAL ;

Trip_BITs_0_to_15 : WORD;
Trip_BITs_16_to_31: WORD;
Trip_BITs_32_to_47: WORD;
Trip_BITs_48_to_63: WORD;
Trip_BITs_64_to_79: WORD;
Trip_BITs_80_to_95: WORD;
Trip_BITs_96_to_121: WORD;
Trip_BITs_122_to_137: WORD;
Trip_BITs_138_to_153: WORD;
Trip_BITs_154_to_169: WORD;
Trip_BITs_170_to_185: WORD;
Trip_BITs_186_to_201: WORD;


Alarm_BITs_0_to_15: WORD;
Alarm_BITs_16_to_31: WORD;
Alarm_BITs_32_to_47: WORD;
Alarm_BITs_48_to_63: WORD;
Alarm_BITs_64_to_79: WORD;
Alarm_BITs_80_to_95: WORD;
Alarm_BITs_96_to_111: WORD;

Status_BITs_0_to_15 : WORD;
Status_BITs_16_to_31 : WORD;
Status_BITs_32_to_47: WORD;
Status_BITs_48_to_63: WORD;
Status_BITs_64_to_79: WORD;
Status_BITs_80_to_95: WORD;
Status_BITs_96_to_111: WORD;
Status_BITs_112_to_127: WORD;




DI_Status_BITs_0_to_15 : WORD;
DI_Status_BITs_16_to_31: WORD;

DO_Status_BITs_16_to_31: WORD;
DO_Status_BITs_32_to_47: WORD;

T_Overload_compressor_motor : BOOL;
T_Compressor_running_failure : BOOL;
T_Low_chilled_medium_outlet : BOOL;
T_Low_sea_water_flow : BOOL;
T_Oil_level_motor_bearing : BOOL;

T_Low_oil_flow : BOOL;
T_Overload_oil_pump_motor : BOOL;
T_Oil_pump_running_failure : BOOL;
T_Low_oil_flow_trip : BOOL;
T_High_temp_oil_receiver : BOOL;
T_Low_temp_oil_receiver : BOOL;
T_Low_suction_pressure : BOOL;
T_High_suction_pressure : BOOL;
T_High_discharge_pressure : BOOL;
T_Low_discharge_pressure : BOOL;
T_High_discharge_temp : BOOL;
T_Low_oil_diff_pressure : BOOL;
T_High_diff_oil_pressure : BOOL;
T_Starting_to_long : BOOL;
T_Surge_detection : BOOL;
T_Comp_thrust_bearing_position : BOOL;
Spare_trip_1 : BOOL;
T_Chilled_pump_run_failure : BOOL;
T_Sea_water_pump_run_failure : BOOL;
T_Low_chilled_medium_flow : BOOL;
T_High_chilled_medium_flow : BOOL;
T_Low_condenser_flow : BOOL;
T_High_condenser_flow : BOOL;
T_Emergency_stop : BOOL;
T_High_comp_mot_DE_bear_temp : BOOL;
T_High_comp_mot_NDE_bear_temp : BOOL;
T_High_motor_air_temp : BOOL;
T_Comp_motor_leak_detection : BOOL;
T_High_comp_mot_DE_bear_vib : BOOL;
T_High_comp_mot_NDE_bear_Vib : BOOL;
T_High_comp_motor_wind_temp : BOOL;
Spare_trip_2 : BOOL;
T_Rotating_stall_trip : BOOL;
T_Analog_inputs : BOOL;
T_Feedback_CW_valve : BOOL;
T_Low_oil_diff_press_prelub : BOOL;
T_Low_oil_diff_press_standstil : BOOL;

T_Spare_3 : BOOL;
T_Spare_4 : BOOL;
T_Spare_5 : BOOL;
T_Spare_6 : BOOL;
T_Spare_7 : BOOL;
T_Spare_8 : BOOL;
T_High_temp_oil_inlet_comp : BOOL;
T_Comp_motor_power_loss : BOOL;
Spare_trip_3 : BOOL;
T_Cathodic_protect_sys_alarm : BOOL;
T_High_oil_filter_diff_press : BOOL;
T_Flow_switch_FT01 : BOOL;
T_Starter_failure_trip : BOOL;
T_Incorrect_feedback_starter_trip : BOOL;

A_VGD_fault : BOOL;
A_High_condenser_flow : BOOL;
A_Rotating_stall : BOOL;
A_High_temp_oil_inlet_comp : BOOL;
SpareAlarm_1 : BOOL;
A_High_motor_air_temp : BOOL;
A_High_control_panel_temp : BOOL;
A_Low_oil_diff_pressure : BOOL;
Spare_alarm_2 : BOOL;
A_High_comp_motor_winding_temp : BOOL;
A_High_comp_mo_DE_bear_temp : BOOL;
A_High_comp_mo_NDE_bear_temp : BOOL;
A_High_comp_mo_DE_bear_vib : BOOL;
A_High_comp_mo_NDE_bear_vib : BOOL;
A_Low_chilled_medium_flow : BOOL;
A_High_chilled_medium_flow : BOOL;
A_Low_sea_water_flow : BOOL;
A_Seawater_pump_not_running : BOOL;
A_Spare : BOOL;
A_Spare_1 : BOOL;
A_Spare_2 : BOOL;
A_Spare_3 : BOOL;
A_Spare_4 : BOOL;
A_Spare_5 : BOOL;
A_Spare_6 : BOOL;
A_Spare_7 : BOOL;
A_Spare_8 : BOOL;
A_Spare_9 : BOOL;
A_Spare_10 : BOOL;
A_Spare_11 : BOOL;
A_High_oil_filter_diff_press : BOOL;
A_Spare_12 : BOOL;
A_Spare_13 : BOOL;
A_Spare_14 : BOOL;
A_Spare_15 : BOOL;
A_Spare_16 : BOOL;
A_Spare_17 : BOOL;
Anti_recycle_status : BOOL;
Low_oil_temperature : BOOL;
Low_oil_temp_auto : BOOL;
Oil_heater : BOOL;
Sea_water_pump : BOOL;
Comp_oil_pump : BOOL;
Bearing_oil_pump : BOOL;
Solenoid_oil_return : BOOL;
Unit_running : BOOL;
Unit_remote : BOOL;
Unit_auto : BOOL;
Unit_manual : BOOL;
Unit_trip : BOOL;
Unit_alarm : BOOL;
Unit_start_switch : BOOL;
Unit_available : BOOL;
Unit_fault : BOOL;
S_Spare_1 : BOOL;
S_Spare_2 : BOOL;
S_Spare_3 : BOOL;
S_Spare_4 : BOOL;
S_Spare_5 : BOOL;
S_Spare_6 : BOOL;
S_Spare_7 : BOOL;
S_Spare_8 : BOOL;
Solenoid_liquid_inj: BOOL;
CW_Flow_ind : BOOL;
Open_chilled_water_valve : BOOL;
Feedback_chilled_water_valve : BOOL;
Open_order_swv_overboard : BOOL;
Close_order_swv_overboard : BOOL;
Open_order_swv_bypass : BOOL;
Close_order_swv_bypass : BOOL;
VFD_man_auto : BOOL ;
VFD_freq_jump_on : BOOL ;
VFD_ramp_100_perc : BOOL ;
VFD_locked_100_perc : BOOL;
VFD_ramp_d_PRVcontrol : BOOL;
PRV_control : BOOL;
VFD_control : BOOL;
VFD_fixed_speed : BOOL;
Spare_151: BOOL;
T_Transformer_winding_temp : BOOL;
A_Transformer_winding_temp : BOOL;
T_trafo_opening_main_breaker : BOOL;
T_VFD : BOOL;
VFD_ready : BOOL;
T_VFD_emergency_stop : BOOL;
T_Low_5VDC_supply : BOOL;
T_High_5VDC_supply : BOOL;
T_Spare_9 : BOOL;
T_Spare_10 : BOOL;
T_Spare_11 : BOOL;
T_Spare_12 : BOOL;
T_Spare_13 : BOOL;
T_Low_liquid_level : BOOL;
T_SW_pump_off_to_long : BOOL;
T_Softstarter_failure : BOOL;
T_Motorstarter_failure : BOOL ;
T_CW_valveopen_failure : BOOL ;
T_SW_valveopen_failure : BOOL ;
T_High_disch_superheat :BOOL ;
T_Low_disch_superheat :BOOL ;
T_High_CW_outlet_temp : BOOL;
T_Low_CW_outlet_temp : BOOL;
T_Low_CW_inlet_temp : BOOL;
T_High_CW_inlet_temp : BOOL;
T_High_SW_outlet_temp : BOOL;
T_Low_SW_outlet_temp : BOOL;
T_Low_SW_inlet_temp : BOOL;
T_High_SW_inlet_temp : BOOL;
T_High_motor_wind_temp_R : BOOL;
T_High_motor_wind_temp_S : BOOL;
T_High_motor_wind_temp_T : BOOL;
T_High_press_ratio : BOOL;
T_Low_press_ratio : BOOL;
T_Low_CW_dP : BOOL;
T_High_CW_dP : BOOL;
T_Low_SW_dP : BOOL;
T_High_SW_dP : BOOL;
T_Long_time_PRV : BOOL;
T_Comp_thrust_neg_move : BOOL;
T_Comp_thrust_pos_move : BOOL;
T_VGD_fault : BOOL;
T_Low_oilpress_prelube : BOOL;
T_Low_temp_oil_inlet_comp : BOOL;
T_Low_oilpress_standby : BOOL;
T_Rotating_stall : BOOL;

T_Sensor_failure_AI_128: BOOL;
T_Sensor_failure_AI_130: BOOL;
T_Sensor_failure_AI_134: BOOL;
T_Sensor_failure_AI_256: BOOL;
T_Sensor_failure_AI_258: BOOL;
T_Sensor_failure_AI_260: BOOL;
T_Sensor_failure_AI_262: BOOL;
T_Sensor_failure_AI_264: BOOL;
T_Sensor_failure_AI_266: BOOL;
T_Sensor_failure_AI_268: BOOL;
T_Sensor_failure_AI_270: BOOL;
T_Sensor_failure_AI_272: BOOL;
T_Sensor_failure_AI_274: BOOL;
T_Sensor_failure_AI_276: BOOL;
T_Sensor_failure_AI_278: BOOL;
T_Sensor_failure_AI_280: BOOL;
T_Sensor_failure_AI_282: BOOL;
T_Sensor_failure_AI_284: BOOL;
T_Sensor_failure_AI_286: BOOL;
T_Sensor_failure_AI_288: BOOL;
T_Sensor_failure_AI_290: BOOL;
T_Sensor_failure_AI_292: BOOL;
T_Sensor_failure_AI_294: BOOL;
T_Sensor_failure_AI_296: BOOL;
T_Sensor_failure_AI_298: BOOL;
T_Sensor_failure_AI_330: BOOL;
T_Sensor_failure_AI_320: BOOL;
T_Sensor_failure_AI_322: BOOL;
T_Sensor_failure_AI_324: BOOL;
T_Sensor_failure_AI_326: BOOL;
T_Sensor_failure_AI_328: BOOL;
T_Sensor_failure_AI_332: BOOL;
T_Sensor_failure_AI_334: BOOL;
T_Sensor_failure_AI_300: BOOL;
T_Sensor_failure_AI_302: BOOL;
T_Sensor_failure_AI_304: BOOL;
T_Sensor_failure_AI_306: BOOL;
T_Sensor_failure_AI_308: BOOL;
T_Sensor_failure_AI_310: BOOL;
T_Sensor_failure_AI_312: BOOL;
T_Sensor_failure_AI_314: BOOL;
T_Sensor_failure_AI_316: BOOL;
T_Sensor_failure_AI_318: BOOL;
T_Sensor_failure_AI_354: BOOL;
T_Sensor_failure_AI_360: BOOL;
T_Sensor_failure_AI_362: BOOL;
T_Sensor_failure_AI_368: BOOL;
T_Sensor_failure_AI_370: BOOL;
T_Sensor_failure_AI_372: BOOL;
T_Sensor_failure_AI_374: BOOL;
T_Sensor_failure_AI_376: BOOL;
T_Sensor_failure_AI_378: BOOL;
T_Sensor_failure_AI_380: BOOL;
T_Sensor_failure_AI_382: BOOL;
T_Sensor_failure_AI_336: BOOL;
T_Sensor_failure_AI_338: BOOL;
T_Sensor_failure_AI_340: BOOL;
T_Sensor_failure_AI_342: BOOL;
T_Sensor_failure_AI_344: BOOL;
T_Sensor_failure_AI_346: BOOL;
T_Sensor_failure_AI_348: BOOL;
T_Sensor_failure_AI_350: BOOL;
T_Sensor_failure_AI_752: BOOL;
T_Sensor_failure_AI_754: BOOL;
T_Sensor_failure_AI_756: BOOL;
T_Sensor_failure_AI_760: BOOL;
T_Sensor_failure_AI_772: BOOL;
T_Sensor_failure_AI_774: BOOL;
T_Sensor_failure_AI_776: BOOL;
T_Sensor_failure_AI_778: BOOL;
T_Sensor_failure_AI_780: BOOL;

A_high_disch_press : BOOL ;
A_low_disch_press : BOOL ;
A_Low_suction_pressure : BOOL;
A_High_suction_pressure : BOOL;
A_High_discharge_temp : BOOL;
A_High_oil_temp_receiver : BOOL;
A_Low_oil_temp_receiver : BOOL;
A_Low_temp_oil_inlet_comp : BOOL;
A_High_oil_diff_pressure : BOOL;
A_Low_discharge_superheat : BOOL;
A_High_discharge_superheat : BOOL;
A_Low_CW_outlet_temp : BOOL;
A_High_CW_outlet_temp : BOOL;
A_Low_CW_inlet_temp : BOOL;
A_High_CW_inlet_temp : BOOL;
A_High_SW_outlet_temp : BOOL;
A_Low_condenser_flow : BOOL;
A_High_press_ratio : BOOL;
A_Low_press_ratio : BOOL;
A_Motor_speed_low : BOOL;
A_Low_SW_outlet_temp : BOOL;
A_Low_SW_inlet_temp : BOOL;
A_High_SW_inlet_temp : BOOL;
A_High_suction_superheat : BOOL;
A_Low_suction_superheat : BOOL;
A_High_temp_oil_separator : BOOL;
A_Low_temp_oil_separator : BOOL;
A_High_motor_wind_temp_R : BOOL;
A_High_motor_wind_temp_S : BOOL;
A_High_motor_wind_temp_T : BOOL;
A_High_CW_dP : BOOL;
A_Low_CW_dP : BOOL;
A_High_SW_dP : BOOL;
A_Low_SW_dP : BOOL;

Start_inhib_time_between_Start : BOOL;
Start_inhib_time_beetween_Stop : BOOL;
Start_inhib_PRV_not_min : BOOL;
Start_inhib_Motor_overload : BOOL;
Remote_bilge_pump_control : BOOL;
CW_pump_running : BOOL;
A_Low_liquid_level : BOOL;
A_Suction_press_limit : BOOL;
A_Discharge_press_limit : BOOL;
A_Discharge_superheat_limit : BOOL;
A_Motor_current_limit : BOOL;


DI_0_0_Emergency_stop : BOOL;
DI_0_0 : BOOL;
DI_0_1 : BOOL;
DI_0_2_Fault_reset : BOOL;
DI_0_2 : BOOL;
DI_0_3 : BOOL;
DI_0_4 : BOOL;
DI_0_5 : BOOL;
DI_0_6_Overload_protection : BOOL;
DI_0_6 : BOOL;
DI_0_7 : BOOL;
DI_1_0_Overload_oilpump : BOOL;
DI_1_0 : BOOL;
DI_1_1 : BOOL;
DI_1_2 : BOOL;
DI_1_3 : BOOL;
Power_available : BOOL;
DI_1_4 : BOOL;
DI_1_5_Starter_failure : BOOL;
DI_1_5 : BOOL;
DI_8_0_Controlpanel_temp : BOOL;
DI_8_0 : BOOL;
DI_8_1 : BOOL;
DI_8_2_VGD_limit_switch : BOOL;
DI_8_2 : BOOL;
DI_8_3_water_leak_motor  : BOOL;
DI_8_3 : BOOL;
DI_8_4_Catodic_protection : BOOL;
DI_8_4 : BOOL;
DI_8_5_Trust_bearing_probe : BOOL;
DI_8_5 : BOOL;
DI_8_6_ESD_operation : BOOL;
DI_8_6 : BOOL;
DI_8_7 : BOOL;
DI_9_0_MV_breaker_available : BOOL;
DI_9_0 : BOOL;
DI_9_1 : BOOL;
DI_9_2_Safe_return_to_port : BOOL;
DI_9_2 : BOOL;
DI_9_3 : BOOL;
DI_9_4_VFD_emergency_stop : BOOL;
DI_9_4 : BOOL;
DI_9_5 : BOOL;
DI_9_6 : BOOL;
DI_9_7 : BOOL;
DO_0_0_Start_signal_comp : BOOL;
DO_0_0 : BOOL;
DO_0_1_Start_signal_oil_pump : BOOL;
DO_0_1 : BOOL;
DO_0_2_Start_signal_SW_pump : BOOL;
DO_0_2 : BOOL;
DO_0_3_Start_signal_CW_pump : BOOL;
DO_0_3 : BOOL;
DO_0_4_Solenoid_valve_oil : BOOL;
DO_0_4 : BOOL;
DO_0_5_Solenoid_valve_liquid : BOOL;
DO_0_5 : BOOL;
DO_0_6_Oil_heater : BOOL;
DO_0_6 : BOOL;
DO_0_7_Comp_heater : BOOL;
DO_0_7 : BOOL;
DO_1_0 : BOOL;
DO_1_1 : BOOL;
DO_8_0_Liquid_valve_open : BOOL;
DO_8_0 : BOOL;
DO_8_1_Liquid_valve_close : BOOL;
DO_8_1 : BOOL;
DO_8_2_VGD_open : BOOL;
DO_8_2 : BOOL;
DO_8_3_VGD_close : BOOL;
DO_8_3 : BOOL;
DO_8_4_PRV_open : BOOL;
DO_8_4 : BOOL;
DO_8_5_PRV_close : BOOL;
DO_8_5 : BOOL;
DO_8_6_HGV_open : BOOL;
DO_8_6 : BOOL;
DO_8_7_HGV_close : BOOL;
DO_8_7 : BOOL;
DO_9_0_Open_order_swv_overboard : BOOL;
DO_9_0 : BOOL;
DO_9_1_Close_order_swv_overboard : BOOL;
DO_9_1 : BOOL;
DO_9_2_Open_order_swv_bypass : BOOL;
DO_9_2 : BOOL;
DO_9_3_Close_order_swv_bypass : BOOL;
DO_9_3 : BOOL;
DO_9_4 : BOOL;
DO_9_5 : BOOL;
DO_9_6 : BOOL;
DO_9_7 : BOOL;
Power_request : BOOL;
DO_12_0 : BOOL;
DO_12_1_Compressor_ready : BOOL;
DO_12_1 : BOOL;
DO_12_2 : BOOL;
DO_12_3 : BOOL;
DO_12_4_Control_panel_alarm : BOOL;
DO_12_4 : BOOL;
DO_12_5_Auto_reset : BOOL;
DO_12_5 : BOOL;
DO_12_6_Unit_running : BOOL;
DO_12_6 : BOOL;
DO_12_7 : BOOL;
Start_inhib_time_Oil_receiver_temp : BOOL;
PrV_in_min : BOOL;



//Graphic variables
Unit_switch_status : INT;
i : INT;
show_trendvalue : ARRAY[0..50] OF BOOL;
select_trendvalue : INT :=0 ;

END_VAR

Temp_chilled_medium_out:=scaleFunction(modbus_var_1000[10],0.1, 0);
Temp_chilled_medium_in:=scaleFunction(modbus_var_1000[11],0.1, 0);
Temp_water_inlet_cond:=scaleFunction(modbus_var_1000[12],0.1, 0);
Press_suction_compr:=scaleFunction(modbus_var_1000[13],0.01, 0);
Press_discharge_compr:=scaleFunction(modbus_var_1000[14],0.01, 0);
Press_oil_receiver:=scaleFunction(modbus_var_1000[15],0.01, 0);
Press_oil_compr:=scaleFunction(modbus_var_1000[16],0.01, 0);
Temp_discharge:=scaleFunction(modbus_var_1000[17],0.1, 0);
Oil_temp_receiver:=scaleFunction(modbus_var_1000[18],0.1, 0);
Max_motor_temp:=scaleFunction(modbus_var_1000[19],0.1, 0);
Temp_motor_bearing_DE:=scaleFunction(modbus_var_1000[20],0.1, 0);
Temp_motor_bearing_NDE:=scaleFunction(modbus_var_1000[21],0.1, 0);
Motor_current:=scaleFunction(modbus_var_1000[22],1.0, 0);
Running_hours_comp_unscaled:=modbus_var_1000[23];
//Anti_recycle_time:=scaleFunction(modbus_var_1000[24],1.0, 0);
Feedback_compressor:=scaleFunction(modbus_var_1000[25],1.0, 0);
Oil_diff_pressure:=scaleFunction(modbus_var_1000[26],0.01, 0);
Suction_saturated_temp:=scaleFunction(modbus_var_1000[27],0.1, 0);
Discharge_saturated_temp:=scaleFunction(modbus_var_1000[28],0.1, 0);
Temp_water_outlet_cond:=scaleFunction(modbus_var_1000[29],0.1, 0);
Temp_motor_wind_R:=scaleFunction(modbus_var_1000[30],0.1, 0);
Temp_motor_wind_S:=scaleFunction(modbus_var_1000[31],0.1, 0);
Temp_motor_wind_T:=scaleFunction(modbus_var_1000[32],0.1, 0);
Temp_motor_air:=scaleFunction(modbus_var_1000[33],0.1, 0);
dP_CW:=scaleFunction(modbus_var_1000[34],0.01, 0);
dP_SW:=scaleFunction(modbus_var_1000[35],0.01, 0);
CW_flow_m3:=scaleFunction(modbus_var_1000[36],1.0, 0);
Temp_oil_inlet_compr:=scaleFunction(modbus_var_1000[37],0.1, 0);
//Stall_detector:=scaleFunction(modbus_var_1000[38],0.01, 0);
SP_CW_controller:=scaleFunction(modbus_var_1000[39],0.1, 0);
Feedback_sea_water_valve:=scaleFunction(modbus_var_1000[40],0.1, 0);
Oil_pressure_before_filter:=scaleFunction(modbus_var_1000[41],0.01, 0);
//Feedback_VGD:=scaleFunction(modbus_var_1000[42],0.1, 0);
Chiller_capacity:=scaleFunction(modbus_var_1000[43],0.1, 0);
Setpoint_oil_pump:=scaleFunction(modbus_var_1000[44],0.01, 0);
Thrust_bearing_position:=scaleFunction(modbus_var_1000[45],0.1, 0);
Oil_pump_running_hours:=scaleFunction(modbus_var_1000[46],10, 0);
Liquid_level_condenser:=scaleFunction(modbus_var_1000[47],0.1, 0);
Oil_Filter_Drop:=scaleFunction(modbus_var_1000[48],0.01, 0);
Proximitor_thrust_pos:=scaleFunction(modbus_var_1000[49],0.1, 0);
//Spare_old_write_bits:=scaleFunction(modbus_var_1000[50],1.0, 0);
Press_chilled_medium_in:=scaleFunction(modbus_var_1000[51],0.01, 0);
Press_water_cond_out:=scaleFunction(modbus_var_1000[52],0.01, 0);
Discharge_superheat:=scaleFunction(modbus_var_1000[53],0.1, 0);
Frequency_oil_pump:=scaleFunction(modbus_var_1000[54],0.1, 0);
Feedback_liquid_valve:=scaleFunction(modbus_var_1000[55],0.1, 0);
Hot_gas_valve_output:=scaleFunction(modbus_var_1000[56],0.1, 0);
Control_signal_unit_d:=scaleFunction(modbus_var_1000[57],0.1, 0);
SP_MC_controller:=scaleFunction(modbus_var_1000[58],0.1, 0);
Prerotary_output:=scaleFunction(modbus_var_1000[59],0.1, 0);
//VGD_output:=scaleFunction(modbus_var_1000[60],0.1, 0);
SP_PID_compressor:=scaleFunction(modbus_var_1000[61],0.1, 0);
Output_PID_suction:=scaleFunction(modbus_var_1000[62],0.1, 0);
Output_PID_discharge:=scaleFunction(modbus_var_1000[63],0.1, 0);
Output_PID_motor:=scaleFunction(modbus_var_1000[64],0.1, 0);
Output_PID_superheat:=scaleFunction(modbus_var_1000[65],0.1, 0);
SP_control:=scaleFunction(modbus_var_1000[66],0.1, 0);
Unit_control_signal:=scaleFunction(modbus_var_1000[67],0.1, 0);
Feedback_PRV:=scaleFunction(modbus_var_1000[68],0.1, 0);
Theta_out:=scaleFunction(modbus_var_1000[69],0.1, 0);
//Alarm_limit_stall_count:=scaleFunction(modbus_var_1000[70],1.0, 0);
//Stall_ramp:=scaleFunction(modbus_var_1000[71],0.1, 0);
//Min_allowed_PRVposition:=scaleFunction(modbus_var_1000[72],0.1, 0);
Number_of_starts:=scaleFunction(modbus_var_1000[73],1.0, 0);
SP_oil_pressure:=scaleFunction(modbus_var_1000[74],0.01, 0);
Setpoint_conv_oil_pump:=scaleFunction(modbus_var_1000[75],0.1, 0);
//Days_above_stall_limit:=scaleFunction(modbus_var_1000[76],1.0, 0);
//Hrs_above_stall_limit:=scaleFunction(modbus_var_1000[77],1.0, 0);
//Min_above_stall_limit:=scaleFunction(modbus_var_1000[78],1.0, 0);
//Sec_above_stall_limit:=scaleFunction(modbus_var_1000[79],1.0, 0);
SP_PID_Level:=scaleFunction(modbus_var_1000[80],0.1, 0);
Control_signal_SW_valve:=scaleFunction(modbus_var_1000[81],0.1, 0);
Feedback_HGV:=scaleFunction(modbus_var_1000[82],0.1, 0);
Liquid_valve_output:=scaleFunction(modbus_var_1000[83],0.1, 0);
SP_PID_seawater:=scaleFunction(modbus_var_1000[84],0.1, 0);
Chiller_capacity_t1:=scaleFunction(modbus_var_1000[85],0.1, 0);
SW_pump_speed_order:=scaleFunction(modbus_var_1000[86],0.1, 0);
Anti_recycle_time:=scaleFunction(modbus_var_1000[87],1.0, 0);
Press_chilled_medium_out:=scaleFunction(modbus_var_1000[88],0.01, 0);
Press_water_cond_inlet:=scaleFunction(modbus_var_1000[89],0.01, 0);
Running_hours_compressormotor:=scaleFunction(modbus_var_1000[90],10, 0);

Trip_BITs_0_to_15:=modbus_var_1000[0];
Trip_BITs_16_to_31:=modbus_var_1000[1];
Trip_BITs_32_to_47:=modbus_var_1000[2];
Trip_BITs_48_to_63:=modbus_var_1000[3];
Trip_BITs_64_to_79:=modbus_var_1000[4];
// Alarm_BITs_80_to_95:=modbus_var_1000[5];
// Alarm_BITs_96_to_111:=modbus_var_1000[6];
Status_BITs_0_to_15:=modbus_var_1000[5];
Status_BITs_16_to_31:=modbus_var_1000[6];


T_Low_suction_pressure:=maskbitFunction(Trip_BITs_0_to_15,0);
T_High_discharge_pressure:=maskbitFunction(Trip_BITs_0_to_15,1);
T_High_discharge_temp:=maskbitFunction(Trip_BITs_0_to_15,2);
T_Low_oil_diff_pressure:=maskbitFunction(Trip_BITs_0_to_15,3);
T_High_diff_oil_pressure:=maskbitFunction(Trip_BITs_0_to_15,4);
T_Starting_to_long:=maskbitFunction(Trip_BITs_0_to_15,5);
T_Surge_detection:=maskbitFunction(Trip_BITs_0_to_15,6);
T_Comp_thrust_bearing_position:=maskbitFunction(Trip_BITs_0_to_15,7);
T_Overload_compressor_motor:=maskbitFunction(Trip_BITs_0_to_15,8);
T_Compressor_running_failure:=maskbitFunction(Trip_BITs_0_to_15,9);
T_Low_chilled_medium_outlet:=maskbitFunction(Trip_BITs_0_to_15,10);
T_Low_oil_flow:=maskbitFunction(Trip_BITs_0_to_15,11);
T_Overload_oil_pump_motor:=maskbitFunction(Trip_BITs_0_to_15,12);
T_Oil_pump_running_failure:=maskbitFunction(Trip_BITs_0_to_15,13);
T_Low_oil_flow_trip:=maskbitFunction(Trip_BITs_0_to_15,14);
T_High_temp_oil_receiver:=maskbitFunction(Trip_BITs_0_to_15,15);
T_High_comp_motor_wind_temp:=maskbitFunction(Trip_BITs_16_to_31,0);
T_High_comp_mot_DE_bear_temp:=maskbitFunction(Trip_BITs_16_to_31,1);
T_High_comp_mot_NDE_bear_temp:=maskbitFunction(Trip_BITs_16_to_31,2);
T_High_motor_air_temp:=maskbitFunction(Trip_BITs_16_to_31,3);
T_Comp_motor_leak_detection:=maskbitFunction(Trip_BITs_16_to_31,4);
T_High_5VDC_supply:=maskbitFunction(Trip_BITs_16_to_31,5);
T_Low_5VDC_supply:=maskbitFunction(Trip_BITs_16_to_31,6);
T_Chilled_pump_run_failure:=maskbitFunction(Trip_BITs_16_to_31,7);
T_Sea_water_pump_run_failure:=maskbitFunction(Trip_BITs_16_to_31,8);
T_Low_chilled_medium_flow:=maskbitFunction(Trip_BITs_16_to_31,9);
T_High_chilled_medium_flow:=maskbitFunction(Trip_BITs_16_to_31,10);
T_Low_sea_water_flow:=maskbitFunction(Trip_BITs_16_to_31,11);
T_High_condenser_flow:=maskbitFunction(Trip_BITs_16_to_31,12);
A_High_temp_oil_inlet_comp:=maskbitFunction(Trip_BITs_16_to_31,13);
T_Comp_motor_power_loss:=maskbitFunction(Trip_BITs_16_to_31,14);
T_Emergency_stop:=maskbitFunction(Trip_BITs_16_to_31,15);
T_Sensor_failure_AI_276:=maskbitFunction(Trip_BITs_32_to_47,0);
T_Sensor_failure_AI_278:=maskbitFunction(Trip_BITs_32_to_47,1);
T_Sensor_failure_AI_280:=maskbitFunction(Trip_BITs_32_to_47,2);
T_Sensor_failure_AI_282:=maskbitFunction(Trip_BITs_32_to_47,3);
T_Sensor_failure_AI_288:=maskbitFunction(Trip_BITs_32_to_47,4);
T_Sensor_failure_AI_292:=maskbitFunction(Trip_BITs_32_to_47,5);
T_Sensor_failure_AI_272:=maskbitFunction(Trip_BITs_32_to_47,6);
T_Sensor_failure_AI_130:=maskbitFunction(Trip_BITs_32_to_47,7);
T_Sensor_failure_AI_134:=maskbitFunction(Trip_BITs_32_to_47,8);
T_Sensor_failure_AI_128:=maskbitFunction(Trip_BITs_32_to_47,9);
T_Sensor_failure_AI_256:=maskbitFunction(Trip_BITs_32_to_47,10);
T_Sensor_failure_AI_274:=maskbitFunction(Trip_BITs_32_to_47,11);
T_Sensor_failure_AI_270:=maskbitFunction(Trip_BITs_32_to_47,12);
T_Sensor_failure_AI_268:=maskbitFunction(Trip_BITs_32_to_47,13);
T_Sensor_failure_AI_286:=maskbitFunction(Trip_BITs_32_to_47,14);
T_Sensor_failure_AI_284:=maskbitFunction(Trip_BITs_32_to_47,15);
T_Sensor_failure_AI_304:=maskbitFunction(Trip_BITs_48_to_63,0);
T_Sensor_failure_AI_308:=maskbitFunction(Trip_BITs_48_to_63,1);
T_Sensor_failure_AI_312:=maskbitFunction(Trip_BITs_48_to_63,2);
T_Sensor_failure_AI_296:=maskbitFunction(Trip_BITs_48_to_63,3);
T_Sensor_failure_AI_300:=maskbitFunction(Trip_BITs_48_to_63,4);
T_Sensor_failure_AI_316:=maskbitFunction(Trip_BITs_48_to_63,5);
T_Sensor_failure_AI_262:=maskbitFunction(Trip_BITs_48_to_63,6);
//T_Sensor_failure_AI_352:=maskbitFunction(Trip_BITs_48_to_63,7);
T_Sensor_failure_AI_354:=maskbitFunction(Trip_BITs_48_to_63,8);
T_Sensor_failure_AI_360:=maskbitFunction(Trip_BITs_48_to_63,9);
T_Sensor_failure_AI_362:=maskbitFunction(Trip_BITs_48_to_63,10);
//T_Sensor_failure_AI_364:=maskbitFunction(Trip_BITs_48_to_63,11);
//T_Rotating_stall_trip:=maskbitFunction(Trip_BITs_48_to_63,12);
T_Analog_inputs:=maskbitFunction(Trip_BITs_48_to_63,13);
T_High_oil_filter_diff_press:=maskbitFunction(Trip_BITs_48_to_63,14);
T_Sensor_failure_AI_260:=maskbitFunction(Trip_BITs_48_to_63,15);
A_High_comp_motor_winding_temp:=maskbitFunction(Trip_BITs_64_to_79,0);
A_High_comp_mo_DE_bear_temp:=maskbitFunction(Trip_BITs_64_to_79,1);
A_High_comp_mo_NDE_bear_temp:=maskbitFunction(Trip_BITs_64_to_79,2);
A_High_motor_air_temp:=maskbitFunction(Trip_BITs_64_to_79,3);
A_Low_chilled_medium_flow:=maskbitFunction(Trip_BITs_64_to_79,4);
A_High_chilled_medium_flow:=maskbitFunction(Trip_BITs_64_to_79,5);
A_Low_sea_water_flow:=maskbitFunction(Trip_BITs_64_to_79,6);
A_High_condenser_flow:=maskbitFunction(Trip_BITs_64_to_79,7);
T_Sensor_failure_AI_258:=maskbitFunction(Trip_BITs_64_to_79,8);
T_Sensor_failure_AI_264:=maskbitFunction(Trip_BITs_64_to_79,9);
T_Sensor_failure_AI_266:=maskbitFunction(Trip_BITs_64_to_79,10);
A_Rotating_stall:=maskbitFunction(Trip_BITs_64_to_79,11);
A_Low_oil_diff_pressure:=maskbitFunction(Trip_BITs_64_to_79,12);
A_High_oil_filter_diff_press:=maskbitFunction(Trip_BITs_64_to_79,13);
A_High_control_panel_temp:=maskbitFunction(Trip_BITs_64_to_79,14);
//A_Spare:=maskbitFunction(Trip_BITs_64_to_79,15);
Unit_running:=maskbitFunction(Status_BITs_0_to_15,0);
Unit_available:=maskbitFunction(Status_BITs_0_to_15,1);
Unit_remote:=maskbitFunction(Status_BITs_0_to_15,2);
Unit_auto:=maskbitFunction(Status_BITs_0_to_15,3);
Anti_recycle_status:=maskbitFunction(Status_BITs_0_to_15,4);
//S_Spare:=maskbitFunction(Status_BITs_0_to_15,5);
//S_Spare:=maskbitFunction(Status_BITs_0_to_15,6);
//S_Spare:=maskbitFunction(Status_BITs_0_to_15,7);
//S_Spare:=maskbitFunction(Status_BITs_0_to_15,8);
Unit_trip:=maskbitFunction(Status_BITs_0_to_15,9);
Unit_alarm:=maskbitFunction(Status_BITs_0_to_15,10);
Unit_fault:=maskbitFunction(Status_BITs_0_to_15,11);
Power_available:=maskbitFunction(Status_BITs_0_to_15,12);
Power_request:=maskbitFunction(Status_BITs_0_to_15,13);
//S_Spare:=maskbitFunction(Status_BITs_0_to_15,14);
PrV_in_min:=maskbitFunction(Status_BITs_0_to_15,15);
Unit_manual:=maskbitFunction(Status_BITs_16_to_31,0);
T_High_temp_oil_inlet_comp:=maskbitFunction(Status_BITs_16_to_31,1);
Unit_start_switch:=maskbitFunction(Status_BITs_16_to_31,2);
Sea_water_pump:=maskbitFunction(Status_BITs_16_to_31,3);

// Graphic controls
IF Unit_remote THEN
	Unit_switch_status:=2;
ELSIF Unit_auto THEN 
	Unit_switch_status:=3;
ELSIF Unit_manual THEN 
	Unit_switch_status:=4;

END_IF ;	

IF select_trendvalue > 0 THEN
	show_trendvalue[select_trendvalue]:= TRUE;
ELSIF select_trendvalue = 0 THEN
	FOR i := 0 TO 50 DO
      show_trendvalue[i] := FALSE;
   	END_FOR
END_IF ;	
	
// timer2 (IN:= TRUE, PT:=T#5S);;
//	IF timer2_Q THEN
//		Temp_motor_bearing_DE := Temp_motor_bearing_DE +1;
//		Motor_current := Motor_current + 1 ;
//		Timer2(IN:= FALSE);
//	END_IF

END_PROGRAM

// Chiller_3
PROGRAM Chiller_3
VAR

timer2 : standard.ton ;
{attribute 'ac_datalog_set_default_group' := 'DatalogChannel_3'}
instStruct : LogStruct;

modbus_var : ARRAY[0..100] OF INT;
modbus_var_1000 : ARRAY[0..123] OF WORD;
modbus_var_1001 : ARRAY[124..247] OF WORD;
modbus_var_1002 : ARRAY[248..371] OF WORD;
{attribute 'ac_datalog_hysteresis' := '0.2'}
{attribute 'ac_datalog' := 'DatalogChannel_3'}
Temp_chilled_medium_out : REAL;
{attribute 'ac_datalog_hysteresis' := '0.2'}
{attribute 'ac_datalog' := 'DatalogChannel_3'}
Temp_chilled_medium_in : REAL;
{attribute 'ac_datalog_hysteresis' := '0.2'}
{attribute 'ac_datalog' := 'DatalogChannel_3'}
Temp_water_inlet_cond : REAL;
{attribute 'ac_datalog_hysteresis' := '0.2'}
{attribute 'ac_datalog' := 'DatalogChannel_3'}
Press_suction_compr : REAL;
{attribute 'ac_datalog_hysteresis' := '0.5'}
{attribute 'ac_datalog' := 'DatalogChannel_3'}
Press_discharge_compr : REAL;
{attribute 'ac_datalog_hysteresis' := '0.5'}
{attribute 'ac_datalog' := 'DatalogChannel_3'}
Press_oil_receiver : REAL;
{attribute 'ac_datalog_hysteresis' := '0.5'}
{attribute 'ac_datalog' := 'DatalogChannel_3'}
Press_oil_compr : REAL;
{attribute 'ac_datalog_hysteresis' := '0.4'}
{attribute 'ac_datalog' := 'DatalogChannel_3'}
Temp_discharge : REAL;
{attribute 'ac_datalog_hysteresis' := '0.5'}
{attribute 'ac_datalog' := 'DatalogChannel_3'}
Oil_temp_receiver : REAL;
{attribute 'ac_datalog_hysteresis' := '0.5'}
{attribute 'ac_datalog' := 'DatalogChannel_3'}
Max_motor_temp : REAL;
{attribute 'ac_datalog_hysteresis' := '0.2'}
{attribute 'ac_datalog' := 'DatalogChannel_3'}
Temp_motor_bearing_DE : REAL;
{attribute 'ac_datalog_hysteresis' := '0.2'}
{attribute 'ac_datalog' := 'DatalogChannel_3'}
Temp_motor_bearing_NDE : REAL;
{attribute 'ac_datalog_hysteresis' := '4'}
{attribute 'ac_datalog' := 'DatalogChannel_3'}
Motor_current : REAL;
{attribute 'ac_datalog_hysteresis' := '50'}
{attribute 'ac_datalog' := 'DatalogChannel_3'}
Running_hours_comp_unscaled : WORD;
{attribute 'ac_datalog_hysteresis' := '50'}
{attribute 'ac_datalog' := 'DatalogChannel_3'}
Running_hours_oil_pump_unscaled : WORD;
{attribute 'ac_datalog' := 'DatalogChannel_3'}
Anti_recycle_time : REAL;
{attribute 'ac_datalog_hysteresis' := '2'}
{attribute 'ac_datalog' := 'DatalogChannel_3'}
Feedback_compressor : REAL;
{attribute 'ac_datalog_hysteresis' := '0.2'}
{attribute 'ac_datalog' := 'DatalogChannel_3'}
Oil_diff_pressure : REAL;
{attribute 'ac_datalog_hysteresis' := '0.3'}
{attribute 'ac_datalog' := 'DatalogChannel_3'}
Suction_saturated_temp : REAL;
{attribute 'ac_datalog_hysteresis' := '0.2'}
{attribute 'ac_datalog' := 'DatalogChannel_3'}
Discharge_saturated_temp : REAL;
{attribute 'ac_datalog_hysteresis' := '0.2'}
{attribute 'ac_datalog' := 'DatalogChannel_3'}
Temp_water_outlet_cond : REAL;
{attribute 'ac_datalog_hysteresis' := '1.0'}
{attribute 'ac_datalog' := 'DatalogChannel_3'}
Temp_motor_wind_R : REAL;
{attribute 'ac_datalog_hysteresis' := '1.0'}
{attribute 'ac_datalog' := 'DatalogChannel_3'}
Temp_motor_wind_S : REAL;
{attribute 'ac_datalog_hysteresis' := '1.0'}
{attribute 'ac_datalog' := 'DatalogChannel_3'}
Temp_motor_wind_T : REAL;
{attribute 'ac_datalog_hysteresis' := '0.2'}
{attribute 'ac_datalog' := 'DatalogChannel_3'}
Temp_motor_air : REAL;
{attribute 'ac_datalog_hysteresis' := '0.04'}
{attribute 'ac_datalog' := 'DatalogChannel_3'}
dP_CW : REAL;
{attribute 'ac_datalog_hysteresis' := '0.04'}
{attribute 'ac_datalog' := 'DatalogChannel_3'}
dP_SW : REAL;
{attribute 'ac_datalog_hysteresis' := '4'}
{attribute 'ac_datalog' := 'DatalogChannel_3'}
Chiller_capacity : REAL;
{attribute 'ac_datalog_hysteresis' := '2'}
{attribute 'ac_datalog' := 'DatalogChannel_3'}
Temp_oil_inlet_compr : REAL;
Spare : REAL;
{attribute 'ac_datalog_hysteresis' := '2'}
{attribute 'ac_datalog' := 'DatalogChannel_3'}
SP_CW_controller : REAL;
{attribute 'ac_datalog_hysteresis' := '2'}
{attribute 'ac_datalog' := 'DatalogChannel_3'}
Setpoint_oil_pump : REAL;
{attribute 'ac_datalog_hysteresis' := '0.02'}
{attribute 'ac_datalog' := 'DatalogChannel_3'}
Thrust_bearing_position : REAL;
{attribute 'ac_datalog_hysteresis' := '50'}
{attribute 'ac_datalog' := 'DatalogChannel_3'}
Oil_pump_running_hours : REAL;
{attribute 'ac_datalog_hysteresis' := '5'}
{attribute 'ac_datalog' := 'DatalogChannel_3'}
Liquid_level_condenser : REAL;
{attribute 'ac_datalog_hysteresis' := '1.0'}
{attribute 'ac_datalog' := 'DatalogChannel_3'}
Oil_Filter_Drop : REAL; 
{attribute 'ac_datalog_hysteresis' := '2'}
{attribute 'ac_datalog' := 'DatalogChannel_3'}
Proximitor_thrust_pos : REAL;
{attribute 'ac_datalog_hysteresis' := '0.4'}
{attribute 'ac_datalog' := 'DatalogChannel_3'}
Press_chilled_medium_in : REAL;
{attribute 'ac_datalog_hysteresis' := '0.2'}
{attribute 'ac_datalog' := 'DatalogChannel_3'}
Press_water_cond_out : REAL;
{attribute 'ac_datalog_hysteresis' := '0.02'}
{attribute 'ac_datalog' := 'DatalogChannel_3'}
Feedback_sea_water_valve : REAL;
{attribute 'ac_datalog_hysteresis' := '1'}
{attribute 'ac_datalog' := 'DatalogChannel_3'}
Oil_pressure_before_filter : REAL;
{attribute 'ac_datalog_hysteresis' := '0.2'}
{attribute 'ac_datalog' := 'DatalogChannel_3'}
Trafo_winding_temp : REAL;
{attribute 'ac_datalog_hysteresis' := '1'}
{attribute 'ac_datalog' := 'DatalogChannel_3'}
Feedback_VGD : REAL;
{attribute 'ac_datalog_hysteresis' := '4'}
{attribute 'ac_datalog' := 'DatalogChannel_3'}
Feedback_liquid_valve : REAL;
{attribute 'ac_datalog_hysteresis' := '3'}
{attribute 'ac_datalog' := 'DatalogChannel_3'}
Feedback_HGV : REAL;
{attribute 'ac_datalog_hysteresis' := '2'}
{attribute 'ac_datalog' := 'DatalogChannel_3'}
Discharge_superheat : REAL;
{attribute 'ac_datalog_hysteresis' := '0.6'}
{attribute 'ac_datalog' := 'DatalogChannel_3'}
Frequency_oil_pump : REAL;
{attribute 'ac_datalog_hysteresis' := '3'}
{attribute 'ac_datalog' := 'DatalogChannel_3'}
Hot_gas_valve_output : REAL;
{attribute 'ac_datalog_hysteresis' := '2'}
{attribute 'ac_datalog' := 'DatalogChannel_3'}
Control_signal_unit_d : REAL;
{attribute 'ac_datalog_hysteresis' := '2'}
{attribute 'ac_datalog' := 'DatalogChannel_3'}
Stall_detector : REAL;
{attribute 'ac_datalog_hysteresis' := '0.2'}
{attribute 'ac_datalog' := 'DatalogChannel_3'}
SP_MC_controller : REAL;
{attribute 'ac_datalog_hysteresis' := '2'}
{attribute 'ac_datalog' := 'DatalogChannel_3'}
Prerotary_output : REAL;
{attribute 'ac_datalog_hysteresis' := '2'}
{attribute 'ac_datalog' := 'DatalogChannel_3'}
VGD_output : REAL;
{attribute 'ac_datalog_hysteresis' := '2'}
{attribute 'ac_datalog' := 'DatalogChannel_3'}
SP_PID_compressor : REAL;
{attribute 'ac_datalog_hysteresis' := '2'}
{attribute 'ac_datalog' := 'DatalogChannel_3'}
Output_PID_suction : REAL;
{attribute 'ac_datalog_hysteresis' := '2'}
{attribute 'ac_datalog' := 'DatalogChannel_3'}
Output_PID_discharge : REAL;
{attribute 'ac_datalog_hysteresis' := '2'}
{attribute 'ac_datalog' := 'DatalogChannel_3'}
Output_PID_motor : REAL;
{attribute 'ac_datalog_hysteresis' := '2'}
{attribute 'ac_datalog' := 'DatalogChannel_3'}
Output_PID_superheat : REAL;
{attribute 'ac_datalog_hysteresis' := '2'}
{attribute 'ac_datalog' := 'DatalogChannel_3'}
SP_control : REAL;
{attribute 'ac_datalog_hysteresis' := '2'}
{attribute 'ac_datalog' := 'DatalogChannel_3'}
Unit_control_signal : REAL;
{attribute 'ac_datalog_hysteresis' := '2'}
{attribute 'ac_datalog' := 'DatalogChannel_3'}
Feedback_PRV : REAL;
{attribute 'ac_datalog_hysteresis' := '0.3'}
{attribute 'ac_datalog' := 'DatalogChannel_3'}
Theta_out : REAL;
{attribute 'ac_datalog_hysteresis' := '50'}
{attribute 'ac_datalog' := 'DatalogChannel_3'}
Alarm_limit_stall_count_unscaled : WORD;
{attribute 'ac_datalog_hysteresis' := '50'}
{attribute 'ac_datalog' := 'DatalogChannel_3'}
Alarm_limit_stall_count : REAL;
{attribute 'ac_datalog_hysteresis' := '2'}
{attribute 'ac_datalog' := 'DatalogChannel_3'}
Stall_ramp : REAL;
Min_allowed_PRVposition : REAL;
Number_of_starts : REAL;
SP_freq_oil_pump_VFD : REAL;
SP_oil_pressure_diff : REAL;
SP_oil_pressure : REAL;
{attribute 'ac_datalog_hysteresis' := '2'}
{attribute 'ac_datalog' := 'DatalogChannel_3'}
Setpoint_conv_oil_pump : REAL;
Days_above_stall_limit : REAL;
Hrs_above_stall_limit : REAL;
Min_above_stall_limit : REAL;
Sec_above_stall_limit : REAL;
{attribute 'ac_datalog_hysteresis' := '2'}
{attribute 'ac_datalog' := 'DatalogChannel_3'}
SP_cond_press : REAL;
{attribute 'ac_datalog_hysteresis' := '2'}
{attribute 'ac_datalog' := 'DatalogChannel_3'}
SP_PID_Level : REAL;
{attribute 'ac_datalog_hysteresis' := '2'}
{attribute 'ac_datalog' := 'DatalogChannel_3'}
Control_signal_SW_valve : REAL;
{attribute 'ac_datalog_hysteresis' := '4'}
{attribute 'ac_datalog' := 'DatalogChannel_3'}
Liquid_valve_output : REAL;
{attribute 'ac_datalog_hysteresis' := '0.2'}
{attribute 'ac_datalog' := 'DatalogChannel_3'}
SP_PID_seawater : REAL;
{attribute 'ac_datalog_hysteresis' := '4'}
{attribute 'ac_datalog' := 'DatalogChannel_3'}
Chiller_capacity_t1 : REAL;
{attribute 'ac_datalog_hysteresis' := '2'}
{attribute 'ac_datalog' := 'DatalogChannel_3'}
SW_pump_speed_order : REAL;
{attribute 'ac_datalog_hysteresis' := '0.4'}
{attribute 'ac_datalog' := 'DatalogChannel_3'}
Press_chilled_medium_out : REAL;
{attribute 'ac_datalog_hysteresis' := '50'}
{attribute 'ac_datalog' := 'DatalogChannel_3'}
Running_hours_compressormotor : REAL;
{attribute 'ac_datalog_hysteresis' := '0.2'}
{attribute 'ac_datalog' := 'DatalogChannel_3'}
Press_water_cond_inlet : REAL;
{attribute 'ac_datalog_hysteresis' := '2'}
{attribute 'ac_datalog' := 'DatalogChannel_3'}
Speed_feedback_VFD : REAL;
{attribute 'ac_datalog_hysteresis' := '2'}
{attribute 'ac_datalog' := 'DatalogChannel_3'}
Order_VFD_perc : REAL;
{attribute 'ac_datalog_hysteresis' := '2'}
{attribute 'ac_datalog' := 'DatalogChannel_3'}
Order_VFD_Hz : REAL;
{attribute 'ac_datalog_hysteresis' := '2'}
{attribute 'ac_datalog' := 'DatalogChannel_3'}
Temp_trafo_wind_U : REAL;
{attribute 'ac_datalog_hysteresis' := '0.2'}
{attribute 'ac_datalog' := 'DatalogChannel_3'}
Temp_trafo_wind_V : REAL;
{attribute 'ac_datalog_hysteresis' := '0.2'}
{attribute 'ac_datalog' := 'DatalogChannel_3'}
Temp_trafo_wind_W : REAL;
{attribute 'ac_datalog_hysteresis' := '2'}
{attribute 'ac_datalog' := 'DatalogChannel_3'}
Opt_speed_VFD_perc : REAL;
{attribute 'ac_datalog_hysteresis' := '2'}
{attribute 'ac_datalog' := 'DatalogChannel_3'}
Opt_speed_VFD_Hz : REAL;
Surge_counter_VFD : REAL;
Spare_4 : REAL;
Spare_3 : REAL;
Spare_2 : REAL;
Spare_0 : REAL;
Vibration_compressor_DE: REAL;
Vibration_compressor_NDE: REAL;
Feedback_seawater_valve_overboard : REAL;
Feedback_seawater_valve_bypass : REAL;
CW_flow_m3: REAL;
SW_flow_m3: REAL;
Max_motor_wind_temp: REAL;
Order_SWW_overboard: REAL;
Order_SWW_bypass: REAL;
{attribute 'ac_datalog_hysteresis' := '0.4'}
{attribute 'ac_datalog' := 'DatalogChannel'}
COP_chiller_mech : REAL ;
{attribute 'ac_datalog_hysteresis' := '50'}
{attribute 'ac_datalog' := 'DatalogChannel'}
P2_mot_1_kW : REAL ;
{attribute 'ac_datalog_hysteresis' := '50'}
{attribute 'ac_datalog' := 'DatalogChannel'}
P1_motor_kW : REAL ;
{attribute 'ac_datalog_hysteresis' := '0.4'}
{attribute 'ac_datalog' := 'DatalogChannel'}
COP_chiller_ele : REAL ;
{attribute 'ac_datalog_hysteresis' := '0.2'}
{attribute 'ac_datalog' := 'DatalogChannel'}
PI_chiller : REAL ;
;{attribute 'ac_datalog_hysteresis' := '40'}
{attribute 'ac_datalog' := 'DatalogChannel'}
Wasted_energy_kW : REAL ;
{attribute 'ac_datalog_hysteresis' := '200'}
{attribute 'ac_datalog' := 'DatalogChannel'}
Chiller_capacity_kW : REAL;
Thrust_bearing_ref_min : REAL ;
Thrust_bearing_ref_max : REAL ;
Thrust_bearing_ref : REAL ;
Q2_chillerMWh : REAL ;
Chiller_P1_MWh : REAL ;
Cal_date_MMYY : REAL ;
Chiller_P2_MWh : REAL ;
Liquid_line_temp : REAL ;
VFD_motor_current : REAL ;
Feedback_liquid_valve_raw : REAL ;
Feedback_VGD_raw : REAL ;
Feedback_PRV_raw : REAL ;
Feedback_HGV_raw : REAL ;
Feedback_seawater_valve_overboard_raw : REAL ;
Feedback_seawater_valve_bypass_raw : REAL ;
SP_cond_press_limit : REAL ;
SP_evap_press_limit : REAL ;
SP_discharge_superheat_limit : REAL ;
SP_t1 : REAL ;
VFD_min_allowed_frequence : REAL ;
VFD_min_allowed_speed : REAL ;

Trip_BITs_0_to_15 : WORD;
Trip_BITs_16_to_31: WORD;
Trip_BITs_32_to_47: WORD;
Trip_BITs_48_to_63: WORD;
Trip_BITs_64_to_79: WORD;
Trip_BITs_80_to_95: WORD;
Trip_BITs_96_to_121: WORD;
Trip_BITs_122_to_137: WORD;
Trip_BITs_138_to_153: WORD;
Trip_BITs_154_to_169: WORD;
Trip_BITs_170_to_185: WORD;
Trip_BITs_186_to_201: WORD;


Alarm_BITs_0_to_15: WORD;
Alarm_BITs_16_to_31: WORD;
Alarm_BITs_32_to_47: WORD;
Alarm_BITs_48_to_63: WORD;
Alarm_BITs_64_to_79: WORD;
Alarm_BITs_80_to_95: WORD;
Alarm_BITs_96_to_111: WORD;

Status_BITs_0_to_15 : WORD;
Status_BITs_16_to_31 : WORD;
Status_BITs_32_to_47: WORD;
Status_BITs_48_to_63: WORD;
Status_BITs_64_to_79: WORD;
Status_BITs_80_to_95: WORD;
Status_BITs_96_to_111: WORD;
Status_BITs_112_to_127: WORD;




DI_Status_BITs_0_to_15 : WORD;
DI_Status_BITs_16_to_31: WORD;

DO_Status_BITs_16_to_31: WORD;
DO_Status_BITs_32_to_47: WORD;

T_Overload_compressor_motor : BOOL;
T_Compressor_running_failure : BOOL;
T_Low_chilled_medium_outlet : BOOL;
T_Low_sea_water_flow : BOOL;
T_Oil_level_motor_bearing : BOOL;

T_Low_oil_flow : BOOL;
T_Overload_oil_pump_motor : BOOL;
T_Oil_pump_running_failure : BOOL;
T_Low_oil_flow_trip : BOOL;
T_High_temp_oil_receiver : BOOL;
T_Low_temp_oil_receiver : BOOL;
T_Low_suction_pressure : BOOL;
T_High_suction_pressure : BOOL;
T_High_discharge_pressure : BOOL;
T_Low_discharge_pressure : BOOL;
T_High_discharge_temp : BOOL;
T_Low_oil_diff_pressure : BOOL;
T_High_diff_oil_pressure : BOOL;
T_Starting_to_long : BOOL;
T_Surge_detection : BOOL;
T_Comp_thrust_bearing_position : BOOL;
Spare_trip_1 : BOOL;
T_Chilled_pump_run_failure : BOOL;
T_Sea_water_pump_run_failure : BOOL;
T_Low_chilled_medium_flow : BOOL;
T_High_chilled_medium_flow : BOOL;
T_Low_condenser_flow : BOOL;
T_High_condenser_flow : BOOL;
T_Emergency_stop : BOOL;
T_High_comp_mot_DE_bear_temp : BOOL;
T_High_comp_mot_NDE_bear_temp : BOOL;
T_High_motor_air_temp : BOOL;
T_Comp_motor_leak_detection : BOOL;
T_High_comp_mot_DE_bear_vib : BOOL;
T_High_comp_mot_NDE_bear_Vib : BOOL;
T_High_comp_motor_wind_temp : BOOL;
Spare_trip_2 : BOOL;
T_Rotating_stall_trip : BOOL;
T_Analog_inputs : BOOL;
T_Feedback_CW_valve : BOOL;
T_Low_oil_diff_press_prelub : BOOL;
T_Low_oil_diff_press_standstil : BOOL;

T_Spare_3 : BOOL;
T_Spare_4 : BOOL;
T_Spare_5 : BOOL;
T_Spare_6 : BOOL;
T_Spare_7 : BOOL;
T_Spare_8 : BOOL;
T_High_temp_oil_inlet_comp : BOOL;
T_Comp_motor_power_loss : BOOL;
Spare_trip_3 : BOOL;
T_Cathodic_protect_sys_alarm : BOOL;
T_High_oil_filter_diff_press : BOOL;
T_Flow_switch_FT01 : BOOL;
T_Starter_failure_trip : BOOL;
T_Incorrect_feedback_starter_trip : BOOL;

A_VGD_fault : BOOL;
A_High_condenser_flow : BOOL;
A_Rotating_stall : BOOL;
A_High_temp_oil_inlet_comp : BOOL;
SpareAlarm_1 : BOOL;
A_High_motor_air_temp : BOOL;
A_High_control_panel_temp : BOOL;
A_Low_oil_diff_pressure : BOOL;
Spare_alarm_2 : BOOL;
A_High_comp_motor_winding_temp : BOOL;
A_High_comp_mo_DE_bear_temp : BOOL;
A_High_comp_mo_NDE_bear_temp : BOOL;
A_High_comp_mo_DE_bear_vib : BOOL;
A_High_comp_mo_NDE_bear_vib : BOOL;
A_Low_chilled_medium_flow : BOOL;
A_High_chilled_medium_flow : BOOL;
A_Low_sea_water_flow : BOOL;
A_Seawater_pump_not_running : BOOL;
A_Spare : BOOL;
A_Spare_1 : BOOL;
A_Spare_2 : BOOL;
A_Spare_3 : BOOL;
A_Spare_4 : BOOL;
A_Spare_5 : BOOL;
A_Spare_6 : BOOL;
A_Spare_7 : BOOL;
A_Spare_8 : BOOL;
A_Spare_9 : BOOL;
A_Spare_10 : BOOL;
A_Spare_11 : BOOL;
A_High_oil_filter_diff_press : BOOL;
A_Spare_12 : BOOL;
A_Spare_13 : BOOL;
A_Spare_14 : BOOL;
A_Spare_15 : BOOL;
A_Spare_16 : BOOL;
A_Spare_17 : BOOL;
Anti_recycle_status : BOOL;
Low_oil_temperature : BOOL;
Low_oil_temp_auto : BOOL;
Oil_heater : BOOL;
Sea_water_pump : BOOL;
Comp_oil_pump : BOOL;
Bearing_oil_pump : BOOL;
Solenoid_oil_return : BOOL;
Unit_running : BOOL;
Unit_remote : BOOL;
Unit_auto : BOOL;
Unit_manual : BOOL;
Unit_trip : BOOL;
Unit_alarm : BOOL;
Unit_start_switch : BOOL;
Unit_available : BOOL;
Unit_fault : BOOL;
S_Spare_1 : BOOL;
S_Spare_2 : BOOL;
S_Spare_3 : BOOL;
S_Spare_4 : BOOL;
S_Spare_5 : BOOL;
S_Spare_6 : BOOL;
S_Spare_7 : BOOL;
S_Spare_8 : BOOL;
Solenoid_liquid_inj: BOOL;
CW_Flow_ind : BOOL;
Open_chilled_water_valve : BOOL;
Feedback_chilled_water_valve : BOOL;
Open_order_swv_overboard : BOOL;
Close_order_swv_overboard : BOOL;
Open_order_swv_bypass : BOOL;
Close_order_swv_bypass : BOOL;
VFD_man_auto : BOOL ;
VFD_freq_jump_on : BOOL ;
VFD_ramp_100_perc : BOOL ;
VFD_locked_100_perc : BOOL;
VFD_ramp_d_PRVcontrol : BOOL;
PRV_control : BOOL;
VFD_control : BOOL;
VFD_fixed_speed : BOOL;
Spare_151: BOOL;
T_Transformer_winding_temp : BOOL;
A_Transformer_winding_temp : BOOL;
T_trafo_opening_main_breaker : BOOL;
T_VFD : BOOL;
VFD_ready : BOOL;
T_VFD_emergency_stop : BOOL;
T_Low_5VDC_supply : BOOL;
T_High_5VDC_supply : BOOL;
T_Spare_9 : BOOL;
T_Spare_10 : BOOL;
T_Spare_11 : BOOL;
T_Spare_12 : BOOL;
T_Spare_13 : BOOL;
T_Low_liquid_level : BOOL;
T_SW_pump_off_to_long : BOOL;
T_Softstarter_failure : BOOL;
T_Motorstarter_failure : BOOL ;
T_CW_valveopen_failure : BOOL ;
T_SW_valveopen_failure : BOOL ;
T_High_disch_superheat :BOOL ;
T_Low_disch_superheat :BOOL ;
T_High_CW_outlet_temp : BOOL;
T_Low_CW_outlet_temp : BOOL;
T_Low_CW_inlet_temp : BOOL;
T_High_CW_inlet_temp : BOOL;
T_High_SW_outlet_temp : BOOL;
T_Low_SW_outlet_temp : BOOL;
T_Low_SW_inlet_temp : BOOL;
T_High_SW_inlet_temp : BOOL;
T_High_motor_wind_temp_R : BOOL;
T_High_motor_wind_temp_S : BOOL;
T_High_motor_wind_temp_T : BOOL;
T_High_press_ratio : BOOL;
T_Low_press_ratio : BOOL;
T_Low_CW_dP : BOOL;
T_High_CW_dP : BOOL;
T_Low_SW_dP : BOOL;
T_High_SW_dP : BOOL;
T_Long_time_PRV : BOOL;
T_Comp_thrust_neg_move : BOOL;
T_Comp_thrust_pos_move : BOOL;
T_VGD_fault : BOOL;
T_Low_oilpress_prelube : BOOL;
T_Low_temp_oil_inlet_comp : BOOL;
T_Low_oilpress_standby : BOOL;
T_Rotating_stall : BOOL;

T_Sensor_failure_AI_128: BOOL;
T_Sensor_failure_AI_130: BOOL;
T_Sensor_failure_AI_134: BOOL;
T_Sensor_failure_AI_256: BOOL;
T_Sensor_failure_AI_258: BOOL;
T_Sensor_failure_AI_260: BOOL;
T_Sensor_failure_AI_262: BOOL;
T_Sensor_failure_AI_264: BOOL;
T_Sensor_failure_AI_266: BOOL;
T_Sensor_failure_AI_268: BOOL;
T_Sensor_failure_AI_270: BOOL;
T_Sensor_failure_AI_272: BOOL;
T_Sensor_failure_AI_274: BOOL;
T_Sensor_failure_AI_276: BOOL;
T_Sensor_failure_AI_278: BOOL;
T_Sensor_failure_AI_280: BOOL;
T_Sensor_failure_AI_282: BOOL;
T_Sensor_failure_AI_284: BOOL;
T_Sensor_failure_AI_286: BOOL;
T_Sensor_failure_AI_288: BOOL;
T_Sensor_failure_AI_290: BOOL;
T_Sensor_failure_AI_292: BOOL;
T_Sensor_failure_AI_294: BOOL;
T_Sensor_failure_AI_296: BOOL;
T_Sensor_failure_AI_298: BOOL;
T_Sensor_failure_AI_330: BOOL;
T_Sensor_failure_AI_320: BOOL;
T_Sensor_failure_AI_322: BOOL;
T_Sensor_failure_AI_324: BOOL;
T_Sensor_failure_AI_326: BOOL;
T_Sensor_failure_AI_328: BOOL;
T_Sensor_failure_AI_332: BOOL;
T_Sensor_failure_AI_334: BOOL;
T_Sensor_failure_AI_300: BOOL;
T_Sensor_failure_AI_302: BOOL;
T_Sensor_failure_AI_304: BOOL;
T_Sensor_failure_AI_306: BOOL;
T_Sensor_failure_AI_308: BOOL;
T_Sensor_failure_AI_310: BOOL;
T_Sensor_failure_AI_312: BOOL;
T_Sensor_failure_AI_314: BOOL;
T_Sensor_failure_AI_316: BOOL;
T_Sensor_failure_AI_318: BOOL;
T_Sensor_failure_AI_352: BOOL;
T_Sensor_failure_AI_354: BOOL;
T_Sensor_failure_AI_360: BOOL;
T_Sensor_failure_AI_362: BOOL;
T_Sensor_failure_AI_364: BOOL;
T_Sensor_failure_AI_368: BOOL;
T_Sensor_failure_AI_370: BOOL;
T_Sensor_failure_AI_372: BOOL;
T_Sensor_failure_AI_374: BOOL;
T_Sensor_failure_AI_376: BOOL;
T_Sensor_failure_AI_378: BOOL;
T_Sensor_failure_AI_380: BOOL;
T_Sensor_failure_AI_382: BOOL;
T_Sensor_failure_AI_336: BOOL;
T_Sensor_failure_AI_338: BOOL;
T_Sensor_failure_AI_340: BOOL;
T_Sensor_failure_AI_342: BOOL;
T_Sensor_failure_AI_344: BOOL;
T_Sensor_failure_AI_346: BOOL;
T_Sensor_failure_AI_348: BOOL;
T_Sensor_failure_AI_350: BOOL;
T_Sensor_failure_AI_752: BOOL;
T_Sensor_failure_AI_754: BOOL;
T_Sensor_failure_AI_756: BOOL;
T_Sensor_failure_AI_760: BOOL;
T_Sensor_failure_AI_772: BOOL;
T_Sensor_failure_AI_774: BOOL;
T_Sensor_failure_AI_776: BOOL;
T_Sensor_failure_AI_778: BOOL;
T_Sensor_failure_AI_780: BOOL;

A_high_disch_press : BOOL ;
A_low_disch_press : BOOL ;
A_Low_suction_pressure : BOOL;
A_High_suction_pressure : BOOL;
A_High_discharge_temp : BOOL;
A_High_oil_temp_receiver : BOOL;
A_Low_oil_temp_receiver : BOOL;
A_Low_temp_oil_inlet_comp : BOOL;
A_High_oil_diff_pressure : BOOL;
A_Low_discharge_superheat : BOOL;
A_High_discharge_superheat : BOOL;
A_Low_CW_outlet_temp : BOOL;
A_High_CW_outlet_temp : BOOL;
A_Low_CW_inlet_temp : BOOL;
A_High_CW_inlet_temp : BOOL;
A_High_SW_outlet_temp : BOOL;
A_Low_condenser_flow : BOOL;
A_High_press_ratio : BOOL;
A_Low_press_ratio : BOOL;
A_Motor_speed_low : BOOL;
A_Low_SW_outlet_temp : BOOL;
A_Low_SW_inlet_temp : BOOL;
A_High_SW_inlet_temp : BOOL;
A_High_suction_superheat : BOOL;
A_Low_suction_superheat : BOOL;
A_High_temp_oil_separator : BOOL;
A_Low_temp_oil_separator : BOOL;
A_High_motor_wind_temp_R : BOOL;
A_High_motor_wind_temp_S : BOOL;
A_High_motor_wind_temp_T : BOOL;
A_High_CW_dP : BOOL;
A_Low_CW_dP : BOOL;
A_High_SW_dP : BOOL;
A_Low_SW_dP : BOOL;

Start_inhib_time_between_Start : BOOL;
Start_inhib_time_beetween_Stop : BOOL;
Start_inhib_PRV_not_min : BOOL;
Start_inhib_Motor_overload : BOOL;
Remote_bilge_pump_control : BOOL;
CW_pump_running : BOOL;
A_Low_liquid_level : BOOL;
A_Suction_press_limit : BOOL;
A_Discharge_press_limit : BOOL;
A_Discharge_superheat_limit : BOOL;
A_Motor_current_limit : BOOL;


DI_0_0_Emergency_stop : BOOL;
DI_0_0 : BOOL;
DI_0_1 : BOOL;
DI_0_2_Fault_reset : BOOL;
DI_0_2 : BOOL;
DI_0_3 : BOOL;
DI_0_4 : BOOL;
DI_0_5 : BOOL;
DI_0_6_Overload_protection : BOOL;
DI_0_6 : BOOL;
DI_0_7 : BOOL;
DI_1_0_Overload_oilpump : BOOL;
DI_1_0 : BOOL;
DI_1_1 : BOOL;
DI_1_2 : BOOL;
DI_1_3 : BOOL;
Power_available : BOOL;
DI_1_4 : BOOL;
DI_1_5_Starter_failure : BOOL;
DI_1_5 : BOOL;
DI_8_0_Controlpanel_temp : BOOL;
DI_8_0 : BOOL;
DI_8_1 : BOOL;
DI_8_2_VGD_limit_switch : BOOL;
DI_8_2 : BOOL;
DI_8_3_water_leak_motor  : BOOL;
DI_8_3 : BOOL;
DI_8_4_Catodic_protection : BOOL;
DI_8_4 : BOOL;
DI_8_5_Trust_bearing_probe : BOOL;
DI_8_5 : BOOL;
DI_8_6_ESD_operation : BOOL;
DI_8_6 : BOOL;
DI_8_7 : BOOL;
DI_9_0_MV_breaker_available : BOOL;
DI_9_0 : BOOL;
DI_9_1 : BOOL;
DI_9_2_Safe_return_to_port : BOOL;
DI_9_2 : BOOL;
DI_9_3 : BOOL;
DI_9_4_VFD_emergency_stop : BOOL;
DI_9_4 : BOOL;
DI_9_5 : BOOL;
DI_9_6 : BOOL;
DI_9_7 : BOOL;
DO_0_0_Start_signal_comp : BOOL;
DO_0_0 : BOOL;
DO_0_1_Start_signal_oil_pump : BOOL;
DO_0_1 : BOOL;
DO_0_2_Start_signal_SW_pump : BOOL;
DO_0_2 : BOOL;
DO_0_3_Start_signal_CW_pump : BOOL;
DO_0_3 : BOOL;
DO_0_4_Solenoid_valve_oil : BOOL;
DO_0_4 : BOOL;
DO_0_5_Solenoid_valve_liquid : BOOL;
DO_0_5 : BOOL;
DO_0_6_Oil_heater : BOOL;
DO_0_6 : BOOL;
DO_0_7_Comp_heater : BOOL;
DO_0_7 : BOOL;
DO_1_0 : BOOL;
DO_1_1 : BOOL;
DO_8_0_Liquid_valve_open : BOOL;
DO_8_0 : BOOL;
DO_8_1_Liquid_valve_close : BOOL;
DO_8_1 : BOOL;
DO_8_2_VGD_open : BOOL;
DO_8_2 : BOOL;
DO_8_3_VGD_close : BOOL;
DO_8_3 : BOOL;
DO_8_4_PRV_open : BOOL;
DO_8_4 : BOOL;
DO_8_5_PRV_close : BOOL;
DO_8_5 : BOOL;
DO_8_6_HGV_open : BOOL;
DO_8_6 : BOOL;
DO_8_7_HGV_close : BOOL;
DO_8_7 : BOOL;
DO_9_0_Open_order_swv_overboard : BOOL;
DO_9_0 : BOOL;
DO_9_1_Close_order_swv_overboard : BOOL;
DO_9_1 : BOOL;
DO_9_2_Open_order_swv_bypass : BOOL;
DO_9_2 : BOOL;
DO_9_3_Close_order_swv_bypass : BOOL;
DO_9_3 : BOOL;
DO_9_4 : BOOL;
DO_9_5 : BOOL;
DO_9_6 : BOOL;
DO_9_7 : BOOL;
Power_request : BOOL;
DO_12_0 : BOOL;
DO_12_1_Compressor_ready : BOOL;
DO_12_1 : BOOL;
DO_12_2 : BOOL;
DO_12_3 : BOOL;
DO_12_4_Control_panel_alarm : BOOL;
DO_12_4 : BOOL;
DO_12_5_Auto_reset : BOOL;
DO_12_5 : BOOL;
DO_12_6_Unit_running : BOOL;
DO_12_6 : BOOL;
DO_12_7 : BOOL;
Start_inhib_time_Oil_receiver_temp : BOOL;
PrV_in_min : BOOL;


//Graphic variables
Unit_switch_status : INT;
i : INT;
show_trendvalue : ARRAY[0..50] OF BOOL;
select_trendvalue : INT :=0 ;

END_VAR


Temp_chilled_medium_out:=scaleFunction(modbus_var_1000[10],0.1, 0);
Temp_chilled_medium_in:=scaleFunction(modbus_var_1000[11],0.1, 0);
Temp_water_inlet_cond:=scaleFunction(modbus_var_1000[12],0.1, 0);
Press_suction_compr:=scaleFunction(modbus_var_1000[13],0.01, 0);
Press_discharge_compr:=scaleFunction(modbus_var_1000[14],0.01, 0);
Press_oil_receiver:=scaleFunction(modbus_var_1000[15],0.01, 0);
Press_oil_compr:=scaleFunction(modbus_var_1000[16],0.01, 0);
Temp_discharge:=scaleFunction(modbus_var_1000[17],0.1, 0);
Oil_temp_receiver:=scaleFunction(modbus_var_1000[18],0.1, 0);
Max_motor_temp:=scaleFunction(modbus_var_1000[19],0.1, 0);
Temp_motor_bearing_DE:=scaleFunction(modbus_var_1000[20],0.1, 0);
Temp_motor_bearing_NDE:=scaleFunction(modbus_var_1000[21],0.1, 0);
Motor_current:=scaleFunction(modbus_var_1000[22],1.0, 0);
Running_hours_comp_unscaled:=modbus_var_1000[23];
//Anti_recycle_time:=scaleFunction(modbus_var_1000[24],1.0, 0);
Feedback_compressor:=scaleFunction(modbus_var_1000[25],1.0, 0);
Oil_diff_pressure:=scaleFunction(modbus_var_1000[26],0.01, 0);
Suction_saturated_temp:=scaleFunction(modbus_var_1000[27],0.1, 0);
Discharge_saturated_temp:=scaleFunction(modbus_var_1000[28],0.1, 0);
Temp_water_outlet_cond:=scaleFunction(modbus_var_1000[29],0.1, 0);
Temp_motor_wind_R:=scaleFunction(modbus_var_1000[30],0.1, 0);
Temp_motor_wind_S:=scaleFunction(modbus_var_1000[31],0.1, 0);
Temp_motor_wind_T:=scaleFunction(modbus_var_1000[32],0.1, 0);
Temp_motor_air:=scaleFunction(modbus_var_1000[33],0.1, 0);
dP_CW:=scaleFunction(modbus_var_1000[34],0.01, 0);
dP_SW:=scaleFunction(modbus_var_1000[35],0.01, 0);
CW_flow_m3:=scaleFunction(modbus_var_1000[36],1.0, 0);
Temp_oil_inlet_compr:=scaleFunction(modbus_var_1000[37],0.1, 0);
Stall_detector:=scaleFunction(modbus_var_1000[38],0.01, 0);
SP_CW_controller:=scaleFunction(modbus_var_1000[39],0.1, 0);
Feedback_sea_water_valve:=scaleFunction(modbus_var_1000[40],0.1, 0);
Oil_pressure_before_filter:=scaleFunction(modbus_var_1000[41],0.01, 0);
Feedback_VGD:=scaleFunction(modbus_var_1000[42],0.1, 0);
Chiller_capacity:=scaleFunction(modbus_var_1000[43],0.1, 0);
Setpoint_oil_pump:=scaleFunction(modbus_var_1000[44],0.01, 0);
Thrust_bearing_position:=scaleFunction(modbus_var_1000[45],0.1, 0);
Oil_pump_running_hours:=scaleFunction(modbus_var_1000[46],10, 0);
Liquid_level_condenser:=scaleFunction(modbus_var_1000[47],0.1, 0);
Oil_Filter_Drop:=scaleFunction(modbus_var_1000[48],0.01, 0);
Proximitor_thrust_pos:=scaleFunction(modbus_var_1000[49],0.1, 0);
//Spare_old_write_bits:=scaleFunction(modbus_var_1000[50],1.0, 0);
Press_chilled_medium_in:=scaleFunction(modbus_var_1000[51],0.01, 0);
Press_water_cond_out:=scaleFunction(modbus_var_1000[52],0.01, 0);
Discharge_superheat:=scaleFunction(modbus_var_1000[53],0.1, 0);
Frequency_oil_pump:=scaleFunction(modbus_var_1000[54],0.1, 0);
Feedback_liquid_valve:=scaleFunction(modbus_var_1000[55],0.1, 0);
Hot_gas_valve_output:=scaleFunction(modbus_var_1000[56],0.1, 0);
Control_signal_unit_d:=scaleFunction(modbus_var_1000[57],0.1, 0);
SP_MC_controller:=scaleFunction(modbus_var_1000[58],0.1, 0);
Prerotary_output:=scaleFunction(modbus_var_1000[59],0.1, 0);
VGD_output:=scaleFunction(modbus_var_1000[60],0.1, 0);
SP_PID_compressor:=scaleFunction(modbus_var_1000[61],0.1, 0);
Output_PID_suction:=scaleFunction(modbus_var_1000[62],0.1, 0);
Output_PID_discharge:=scaleFunction(modbus_var_1000[63],0.1, 0);
Output_PID_motor:=scaleFunction(modbus_var_1000[64],0.1, 0);
Output_PID_superheat:=scaleFunction(modbus_var_1000[65],0.1, 0);
SP_control:=scaleFunction(modbus_var_1000[66],0.1, 0);
Unit_control_signal:=scaleFunction(modbus_var_1000[67],0.1, 0);
Feedback_PRV:=scaleFunction(modbus_var_1000[68],0.1, 0);
Theta_out:=scaleFunction(modbus_var_1000[69],0.1, 0);
Alarm_limit_stall_count:=scaleFunction(modbus_var_1000[70],1.0, 0);
Stall_ramp:=scaleFunction(modbus_var_1000[71],0.1, 0);
Min_allowed_PRVposition:=scaleFunction(modbus_var_1000[72],0.1, 0);
Number_of_starts:=scaleFunction(modbus_var_1000[73],1.0, 0);
SP_oil_pressure:=scaleFunction(modbus_var_1000[74],0.01, 0);
Setpoint_conv_oil_pump:=scaleFunction(modbus_var_1000[75],0.1, 0);
Days_above_stall_limit:=scaleFunction(modbus_var_1000[76],1.0, 0);
Hrs_above_stall_limit:=scaleFunction(modbus_var_1000[77],1.0, 0);
Min_above_stall_limit:=scaleFunction(modbus_var_1000[78],1.0, 0);
Sec_above_stall_limit:=scaleFunction(modbus_var_1000[79],1.0, 0);
SP_PID_Level:=scaleFunction(modbus_var_1000[80],0.1, 0);
Control_signal_SW_valve:=scaleFunction(modbus_var_1000[81],0.1, 0);
Feedback_HGV:=scaleFunction(modbus_var_1000[82],0.1, 0);
Liquid_valve_output:=scaleFunction(modbus_var_1000[83],0.1, 0);
SP_PID_seawater:=scaleFunction(modbus_var_1000[84],0.1, 0);
Chiller_capacity_t1:=scaleFunction(modbus_var_1000[85],0.1, 0);
SW_pump_speed_order:=scaleFunction(modbus_var_1000[86],0.1, 0);
Anti_recycle_time:=scaleFunction(modbus_var_1000[87],1.0, 0);
Press_chilled_medium_out:=scaleFunction(modbus_var_1000[88],0.01, 0);
Press_water_cond_inlet:=scaleFunction(modbus_var_1000[89],0.01, 0);
Running_hours_compressormotor:=scaleFunction(modbus_var_1000[90],10, 0);

Trip_BITs_0_to_15:=modbus_var_1000[0];
Trip_BITs_16_to_31:=modbus_var_1000[1];
Trip_BITs_32_to_47:=modbus_var_1000[2];
Trip_BITs_48_to_63:=modbus_var_1000[3];
Trip_BITs_64_to_79:=modbus_var_1000[4];
// Alarm_BITs_80_to_95:=modbus_var_1000[5];
// Alarm_BITs_96_to_111:=modbus_var_1000[6];
Status_BITs_0_to_15:=modbus_var_1000[5];
Status_BITs_16_to_31:=modbus_var_1000[6];

T_Low_suction_pressure:=maskbitFunction(Trip_BITs_0_to_15,0);
T_High_discharge_pressure:=maskbitFunction(Trip_BITs_0_to_15,1);
T_High_discharge_temp:=maskbitFunction(Trip_BITs_0_to_15,2);
T_Low_oil_diff_pressure:=maskbitFunction(Trip_BITs_0_to_15,3);
T_High_diff_oil_pressure:=maskbitFunction(Trip_BITs_0_to_15,4);
T_Starting_to_long:=maskbitFunction(Trip_BITs_0_to_15,5);
T_Surge_detection:=maskbitFunction(Trip_BITs_0_to_15,6);
T_Comp_thrust_bearing_position:=maskbitFunction(Trip_BITs_0_to_15,7);
T_Overload_compressor_motor:=maskbitFunction(Trip_BITs_0_to_15,8);
T_Compressor_running_failure:=maskbitFunction(Trip_BITs_0_to_15,9);
T_Low_chilled_medium_outlet:=maskbitFunction(Trip_BITs_0_to_15,10);
T_Low_oil_flow:=maskbitFunction(Trip_BITs_0_to_15,11);
T_Overload_oil_pump_motor:=maskbitFunction(Trip_BITs_0_to_15,12);
T_Oil_pump_running_failure:=maskbitFunction(Trip_BITs_0_to_15,13);
T_Low_oil_flow_trip:=maskbitFunction(Trip_BITs_0_to_15,14);
T_High_temp_oil_receiver:=maskbitFunction(Trip_BITs_0_to_15,15);
T_High_comp_motor_wind_temp:=maskbitFunction(Trip_BITs_16_to_31,0);
T_High_comp_mot_DE_bear_temp:=maskbitFunction(Trip_BITs_16_to_31,1);
T_High_comp_mot_NDE_bear_temp:=maskbitFunction(Trip_BITs_16_to_31,2);
T_High_motor_air_temp:=maskbitFunction(Trip_BITs_16_to_31,3);
T_Comp_motor_leak_detection:=maskbitFunction(Trip_BITs_16_to_31,4);
T_High_5VDC_supply:=maskbitFunction(Trip_BITs_16_to_31,5);
T_Low_5VDC_supply:=maskbitFunction(Trip_BITs_16_to_31,6);
T_Chilled_pump_run_failure:=maskbitFunction(Trip_BITs_16_to_31,7);
T_Sea_water_pump_run_failure:=maskbitFunction(Trip_BITs_16_to_31,8);
T_Low_chilled_medium_flow:=maskbitFunction(Trip_BITs_16_to_31,9);
T_High_chilled_medium_flow:=maskbitFunction(Trip_BITs_16_to_31,10);
T_Low_sea_water_flow:=maskbitFunction(Trip_BITs_16_to_31,11);
T_High_condenser_flow:=maskbitFunction(Trip_BITs_16_to_31,12);
A_High_temp_oil_inlet_comp:=maskbitFunction(Trip_BITs_16_to_31,13);
T_Comp_motor_power_loss:=maskbitFunction(Trip_BITs_16_to_31,14);
T_Emergency_stop:=maskbitFunction(Trip_BITs_16_to_31,15);
T_Sensor_failure_AI_276:=maskbitFunction(Trip_BITs_32_to_47,0);
T_Sensor_failure_AI_278:=maskbitFunction(Trip_BITs_32_to_47,1);
T_Sensor_failure_AI_280:=maskbitFunction(Trip_BITs_32_to_47,2);
T_Sensor_failure_AI_282:=maskbitFunction(Trip_BITs_32_to_47,3);
T_Sensor_failure_AI_288:=maskbitFunction(Trip_BITs_32_to_47,4);
T_Sensor_failure_AI_292:=maskbitFunction(Trip_BITs_32_to_47,5);
T_Sensor_failure_AI_272:=maskbitFunction(Trip_BITs_32_to_47,6);
T_Sensor_failure_AI_130:=maskbitFunction(Trip_BITs_32_to_47,7);
T_Sensor_failure_AI_134:=maskbitFunction(Trip_BITs_32_to_47,8);
T_Sensor_failure_AI_128:=maskbitFunction(Trip_BITs_32_to_47,9);
T_Sensor_failure_AI_256:=maskbitFunction(Trip_BITs_32_to_47,10);
T_Sensor_failure_AI_274:=maskbitFunction(Trip_BITs_32_to_47,11);
T_Sensor_failure_AI_270:=maskbitFunction(Trip_BITs_32_to_47,12);
T_Sensor_failure_AI_268:=maskbitFunction(Trip_BITs_32_to_47,13);
T_Sensor_failure_AI_286:=maskbitFunction(Trip_BITs_32_to_47,14);
T_Sensor_failure_AI_284:=maskbitFunction(Trip_BITs_32_to_47,15);
T_Sensor_failure_AI_304:=maskbitFunction(Trip_BITs_48_to_63,0);
T_Sensor_failure_AI_308:=maskbitFunction(Trip_BITs_48_to_63,1);
T_Sensor_failure_AI_312:=maskbitFunction(Trip_BITs_48_to_63,2);
T_Sensor_failure_AI_296:=maskbitFunction(Trip_BITs_48_to_63,3);
T_Sensor_failure_AI_300:=maskbitFunction(Trip_BITs_48_to_63,4);
T_Sensor_failure_AI_316:=maskbitFunction(Trip_BITs_48_to_63,5);
T_Sensor_failure_AI_262:=maskbitFunction(Trip_BITs_48_to_63,6);
T_Sensor_failure_AI_352:=maskbitFunction(Trip_BITs_48_to_63,7);
T_Sensor_failure_AI_354:=maskbitFunction(Trip_BITs_48_to_63,8);
T_Sensor_failure_AI_360:=maskbitFunction(Trip_BITs_48_to_63,9);
T_Sensor_failure_AI_362:=maskbitFunction(Trip_BITs_48_to_63,10);
T_Sensor_failure_AI_364:=maskbitFunction(Trip_BITs_48_to_63,11);
T_Rotating_stall_trip:=maskbitFunction(Trip_BITs_48_to_63,12);
T_Analog_inputs:=maskbitFunction(Trip_BITs_48_to_63,13);
T_High_oil_filter_diff_press:=maskbitFunction(Trip_BITs_48_to_63,14);
T_Sensor_failure_AI_260:=maskbitFunction(Trip_BITs_48_to_63,15);
A_High_comp_motor_winding_temp:=maskbitFunction(Trip_BITs_64_to_79,0);
A_High_comp_mo_DE_bear_temp:=maskbitFunction(Trip_BITs_64_to_79,1);
A_High_comp_mo_NDE_bear_temp:=maskbitFunction(Trip_BITs_64_to_79,2);
A_High_motor_air_temp:=maskbitFunction(Trip_BITs_64_to_79,3);
A_Low_chilled_medium_flow:=maskbitFunction(Trip_BITs_64_to_79,4);
A_High_chilled_medium_flow:=maskbitFunction(Trip_BITs_64_to_79,5);
A_Low_sea_water_flow:=maskbitFunction(Trip_BITs_64_to_79,6);
A_High_condenser_flow:=maskbitFunction(Trip_BITs_64_to_79,7);
T_Sensor_failure_AI_258:=maskbitFunction(Trip_BITs_64_to_79,8);
T_Sensor_failure_AI_264:=maskbitFunction(Trip_BITs_64_to_79,9);
T_Sensor_failure_AI_266:=maskbitFunction(Trip_BITs_64_to_79,10);
A_Rotating_stall:=maskbitFunction(Trip_BITs_64_to_79,11);
A_Low_oil_diff_pressure:=maskbitFunction(Trip_BITs_64_to_79,12);
A_High_oil_filter_diff_press:=maskbitFunction(Trip_BITs_64_to_79,13);
A_High_control_panel_temp:=maskbitFunction(Trip_BITs_64_to_79,14);
//A_Spare:=maskbitFunction(Trip_BITs_64_to_79,15);
Unit_running:=maskbitFunction(Status_BITs_0_to_15,0);
Unit_available:=maskbitFunction(Status_BITs_0_to_15,1);
Unit_remote:=maskbitFunction(Status_BITs_0_to_15,2);
Unit_auto:=maskbitFunction(Status_BITs_0_to_15,3);
Anti_recycle_status:=maskbitFunction(Status_BITs_0_to_15,4);
//S_Spare:=maskbitFunction(Status_BITs_0_to_15,5);
//S_Spare:=maskbitFunction(Status_BITs_0_to_15,6);
//S_Spare:=maskbitFunction(Status_BITs_0_to_15,7);
//S_Spare:=maskbitFunction(Status_BITs_0_to_15,8);
Unit_trip:=maskbitFunction(Status_BITs_0_to_15,9);
Unit_alarm:=maskbitFunction(Status_BITs_0_to_15,10);
Unit_fault:=maskbitFunction(Status_BITs_0_to_15,11);
Power_available:=maskbitFunction(Status_BITs_0_to_15,12);
Power_request:=maskbitFunction(Status_BITs_0_to_15,13);
//S_Spare:=maskbitFunction(Status_BITs_0_to_15,14);
PrV_in_min:=maskbitFunction(Status_BITs_0_to_15,15);
Unit_manual:=maskbitFunction(Status_BITs_16_to_31,0);
T_High_temp_oil_inlet_comp:=maskbitFunction(Status_BITs_16_to_31,1);
Unit_start_switch:=maskbitFunction(Status_BITs_16_to_31,2);
Sea_water_pump:=maskbitFunction(Status_BITs_16_to_31,3);


// Graphic controls
IF Unit_remote THEN
	Unit_switch_status:=2;
ELSIF Unit_auto THEN 
	Unit_switch_status:=3;
ELSIF Unit_manual THEN 
	Unit_switch_status:=4;

END_IF ;	

IF select_trendvalue > 0 THEN
	show_trendvalue[select_trendvalue]:= TRUE;
ELSIF select_trendvalue = 0 THEN
	FOR i := 0 TO 50 DO
      show_trendvalue[i] := FALSE;
   	END_FOR
END_IF ;	
	
// timer2 (IN:= TRUE, PT:=T#5S);;
//	IF timer2_Q THEN
//		Temp_motor_bearing_DE := Temp_motor_bearing_DE +1;
//		Motor_current := Motor_current + 1 ;
//		Timer2(IN:= FALSE);
//	END_IF

END_PROGRAM

// Chiller_4
PROGRAM Chiller_4
VAR

timer2 : standard.ton ;
{attribute 'ac_datalog_set_default_group' := 'DatalogChannel_4'}
instStruct : LogStruct;

